REGION Network 6
   RUNG wire#powerrail
      Contact( #calcula )
      wire#w1
      { S7_Templates := "SrcType := Real"; S7_GenerateENO := "TRUE" } Sub(in1 := #FATOR, in2 := #SETPOINT, out => #FATOR)
   END_RUNG
   RUNG wire#w1
      { S7_Templates := "SrcType := Real"; S7_GenerateENO := "TRUE" } Div(in1 := #FATOR, in2 := #SETPOINT, out => #FATOR)
   END_RUNG
   RUNG wire#w1
      { S7_Templates := "SrcType := Real"; S7_GenerateENO := "TRUE" } Mul(in1 := #FATOR, in2 := #COR_MAX, out => #FATOR)
      { S7_Templates := "SrcType := Real"; S7_GenerateENO := "TRUE" } Mul(in1 := #FATOR, in2 := 0.01, out => #FATOR)
      { S7_Templates := "SrcType := Real"; S7_GenerateENO := "TRUE" } Mul(in1 := #FATOR, in2 := #VELOCIDADE_BASE, out => #CORRECAO)
   END_RUNG
   // the same network as SCL:
   // ENO of a box is taken as its EN; it also drops when the box reports an error
   IF #calcula THEN
       #FATOR := #FATOR - #SETPOINT;
       #FATOR := #FATOR / #SETPOINT;
       #FATOR := #FATOR * #COR_MAX;
       #FATOR := #FATOR * 0.01;
       #CORRECAO := #FATOR * #VELOCIDADE_BASE;
   END_IF;
END_REGION
END_FUNCTION_BLOCK

FUNCTION "GRUPO1" : Void   // FC2, LAD
{ S7_Optimized_Access := 'FALSE' }
VERSION : 0.1
   VAR_TEMP
      RASQ_R : Real;
      RASQ_DI : DInt;
      RASQ_R2 : Real;
   END_VAR
   VAR_TEMP   // added for the SCL form of the ladder/FBD networks
      _w1 : Bool;
      _w2 : Bool;
      _w3 : Bool;
      _w4 : Bool;
      _w5 : Bool;
      _w6 : Bool;
      _w7 : Bool;
      _w8 : Bool;
   END_VAR
BEGIN

REGION Network 1: RESET ALARMES
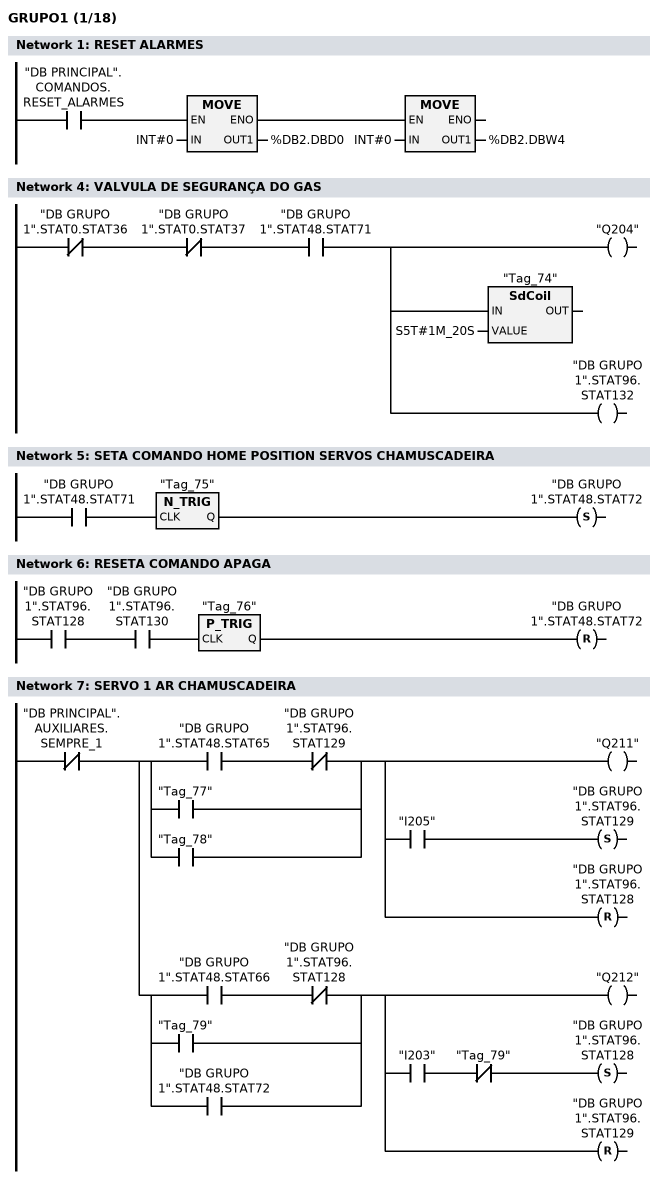
   RUNG wire#powerrail
      Contact( "DB PRINCIPAL".COMANDOS.RESET_ALARMES )
      { S7_GenerateENO := "TRUE" } Move(in := INT#0, out1 => %DB2.DBD0)
      { S7_GenerateENO := "TRUE" } Move(in := INT#0, out1 => %DB2.DBW4)
   END_RUNG
   // the same network as SCL:
   // ENO of a box is taken as its EN; it also drops when the box reports an error
   IF "DB PRINCIPAL".COMANDOS.RESET_ALARMES THEN
       %DB2.DBD0 := INT#0;
       %DB2.DBW4 := INT#0;
   END_IF;
END_REGION

REGION Network 2 (STL): TERMICOS
         A     "DB PRINCIPAL".AUXILIARES.SEMPRE_1;
         S     <??.?>;
         A     <??.?>;
         A     "I102";
         S     "DB GRUPO 1".STAT0.STAT5;
         A     <??.?>;
         A     "I103";
         S     "DB GRUPO 1".STAT0.STAT6;
         A     <??.?>;
         A     "I104";
         S     "DB GRUPO 1".STAT0.STAT7;
         A     <??.?>;
         A     "I105";
         S     "DB GRUPO 1".STAT0.STAT8;
         A     <??.?>;
         A     "I107";
         S     "DB GRUPO 1".STAT0.STAT17;
         A     <??.?>;
         A     "I110";
         S     "DB GRUPO 1".STAT0.STAT18;
         A     <??.?>;
         A     "I122";
         S     "DB GRUPO 1".STAT0.STAT19;
         A     <??.?>;
         A     "I123";
         S     "DB GRUPO 1".STAT0.STAT20;
         A     <??.?>;
         AN    "I124";
         A     "DB GRUPO 1".STAT48.STAT71;
         S     "DB GRUPO 1".STAT0.STAT3;
         A     <??.?>;
         AN    "I125";
         A     "DB GRUPO 1".STAT48.STAT71;
         S     "DB GRUPO 1".STAT0.STAT4;
         A     <??.?>;
         A     "I126";
         S     "DB GRUPO 1".STAT0.STAT10;
         A     <??.?>;
         A     "I127";
         S     "DB GRUPO 1".STAT0.STAT11;
         A     <??.?>;
         A     "I131";
         S     "DB GRUPO 1".STAT0.STAT21;
         A     <??.?>;
         A     "I133";
         S     "DB GRUPO 1".STAT0.STAT22;
         A     <??.?>;
         A     "I135";
         S     "DB GRUPO 1".STAT0.STAT23;
         A     <??.?>;
         A     "I137";
         S     "DB GRUPO 1".STAT0.STAT24;
         A     <??.?>;
         A     "I106";
         A     "DB GRUPO 1".STAT48.STAT71;
         S     "DB GRUPO 1".STAT0.STAT9;
         A     <??.?>;
         AN    "I322";
         S     "DB GRUPO 1".STAT0.STAT25;
END_REGION

REGION Network 3 (STL): ALARMES CHAMUSCADEIRA
         A     "DB GRUPO 1".STAT48.STAT71;
         =     <??.?>;
         A     <??.?>;
         AN    "I200";
         A     "Tag_72";
         S     "DB GRUPO 1".STAT0.STAT33;
         A     <??.?>;
         AN    "I207";
         A     "Tag_73";
         S     "DB GRUPO 1".STAT0.STAT38;
         A     <??.?>;
         AN    "I201";
         S     "DB GRUPO 1".STAT0.STAT34;
         A     <??.?>;
         A     "I202";
         A     "Tag_74";
         S     "DB GRUPO 1".STAT0.STAT35;
         A     <??.?>;
         AN    "I204";
         S     "DB GRUPO 1".STAT0.STAT36;
         A     <??.?>;
         A     "DB PRINCIPAL".AUXILIARES.SEMPRE_0;
         AN    "I206";
         S     "DB GRUPO 1".STAT0.STAT37;
         A     <??.?>;
         A(;
         L     "DB GRUPO 1".STAT154.STAT162;
         L     "DB GRUPO 1".STAT138.STAT146;
         >R;
         );
         S     "DB GRUPO 1".STAT0.STAT39;
         A     <??.?>;
         A(;
         L     "DB GRUPO 1".STAT154.STAT163;
         L     "DB GRUPO 1".STAT138.STAT147;
         >R;
         );
         S     "DB GRUPO 1".STAT0.STAT40;
         A     <??.?>;
         A(;
         L     "DB GRUPO 1".STAT154.STAT164;
         L     "DB GRUPO 1".STAT138.STAT148;
         >R;
         );
         S     "DB GRUPO 1".STAT0.STAT41;
         A     <??.?>;
         A(;
         L     "DB GRUPO 1".STAT154.STAT165;
         L     "DB GRUPO 1".STAT138.STAT149;
         >R;
         );
         S     "DB GRUPO 1".STAT0.STAT42;
         A     <??.?>;
         A     "I214";
         S     "DB GRUPO 1".STAT0.STAT43;
         A     <??.?>;
         A     "I215";
         S     "DB GRUPO 1".STAT0.STAT44;
         A     <??.?>;
         A     "I216";
         S     "DB GRUPO 1".STAT0.STAT45;
         A     <??.?>;
         A     "I217";
         S     "DB GRUPO 1".STAT0.STAT46;
         NOP   0;
END_REGION

REGION Network 4: VALVULA DE SEGURANÇA DO GAS
   // no SCL statement known for SdCoil: written as a call
   "Q204" := NOT "DB GRUPO 1".STAT0.STAT36 AND NOT "DB GRUPO 1".STAT0.STAT37 AND "DB GRUPO 1".STAT48.STAT71;
   #_w1 := "Q204";
   SdCoil(value := S5T#1M_20S, operand := "Tag_74", in := "Q204");
   "DB GRUPO 1".STAT96.STAT132 := #_w1;
END_REGION

REGION Network 5: SETA COMANDO HOME POSITION SERVOS CHAMUSCADEIRA
   RUNG wire#powerrail
      Contact( "DB GRUPO 1".STAT48.STAT71 )
      N_Trig( "Tag_75" )
      S_Coil( "DB GRUPO 1".STAT48.STAT72 )
   END_RUNG
   // the same network as SCL:
   #_w1 := NOT "DB GRUPO 1".STAT48.STAT71 AND "Tag_75";   // falling edge
   "Tag_75" := "DB GRUPO 1".STAT48.STAT71;
   IF #_w1 THEN "DB GRUPO 1".STAT48.STAT72 := TRUE; END_IF;
END_REGION

REGION Network 6: RESETA COMANDO APAGA
   RUNG wire#powerrail
      Contact( "DB GRUPO 1".STAT96.STAT128 )
      Contact( "DB GRUPO 1".STAT96.STAT130 )
      P_Trig( "Tag_76" )
      R_Coil( "DB GRUPO 1".STAT48.STAT72 )
   END_RUNG
   // the same network as SCL:
   #_w1 := "DB GRUPO 1".STAT96.STAT128 AND "DB GRUPO 1".STAT96.STAT130;
   #_w2 := #_w1 AND NOT "Tag_76";   // rising edge
   "Tag_76" := #_w1;
   IF #_w2 THEN "DB GRUPO 1".STAT48.STAT72 := FALSE; END_IF;
END_REGION

REGION Network 7: SERVO 1 AR CHAMUSCADEIRA
   RUNG wire#powerrail
      I_Contact( "DB PRINCIPAL".AUXILIARES.SEMPRE_1 )
      wire#w1
      Contact( "DB GRUPO 1".STAT48.STAT65 )
      I_Contact( "DB GRUPO 1".STAT96.STAT129 )
      wire#w2
      Coil( "Q211" )
   END_RUNG
   RUNG wire#w1
      Contact( "Tag_77" )
   END_RUNG wire#w2
   RUNG wire#w1
      Contact( "Tag_78" )
   END_RUNG wire#w2
   RUNG wire#w2
      Contact( "I205" )
      S_Coil( "DB GRUPO 1".STAT96.STAT129 )
   END_RUNG
   RUNG wire#w2
      R_Coil( "DB GRUPO 1".STAT96.STAT128 )
   END_RUNG
   RUNG wire#w1
      Contact( "DB GRUPO 1".STAT48.STAT66 )
      I_Contact( "DB GRUPO 1".STAT96.STAT128 )
      wire#w3
      Coil( "Q212" )
   END_RUNG
   RUNG wire#w1
      Contact( "Tag_79" )
   END_RUNG wire#w3
   RUNG wire#w1
      Contact( "DB GRUPO 1".STAT48.STAT72 )
   END_RUNG wire#w3
   RUNG wire#w3
      Contact( "I203" )
      I_Contact( "Tag_79" )
      S_Coil( "DB GRUPO 1".STAT96.STAT128 )
   END_RUNG
   RUNG wire#w3
      R_Coil( "DB GRUPO 1".STAT96.STAT129 )
   END_RUNG
   // the same network as SCL:
   #_w1 := NOT "DB PRINCIPAL".AUXILIARES.SEMPRE_1;
   "Q211" := #_w1 AND (("DB GRUPO 1".STAT48.STAT65 AND NOT "DB GRUPO 1".STAT96.STAT129) OR "Tag_77" OR "Tag_78");
   IF "Q211" AND "I205" THEN "DB GRUPO 1".STAT96.STAT129 := TRUE; END_IF;
   IF "Q211" THEN "DB GRUPO 1".STAT96.STAT128 := FALSE; END_IF;
   "Q212" := #_w1 AND (("DB GRUPO 1".STAT48.STAT66 AND NOT "DB GRUPO 1".STAT96.STAT128) OR "Tag_79" OR "DB GRUPO 1".STAT48.STAT72);
   IF "Q212" AND "I203" AND NOT "Tag_79" THEN "DB GRUPO 1".STAT96.STAT128 := TRUE; END_IF;
   IF "Q212" THEN "DB GRUPO 1".STAT96.STAT129 := FALSE; END_IF;
END_REGION

REGION Network 8: SERVO 2 AR CHAMUSCADEIRA
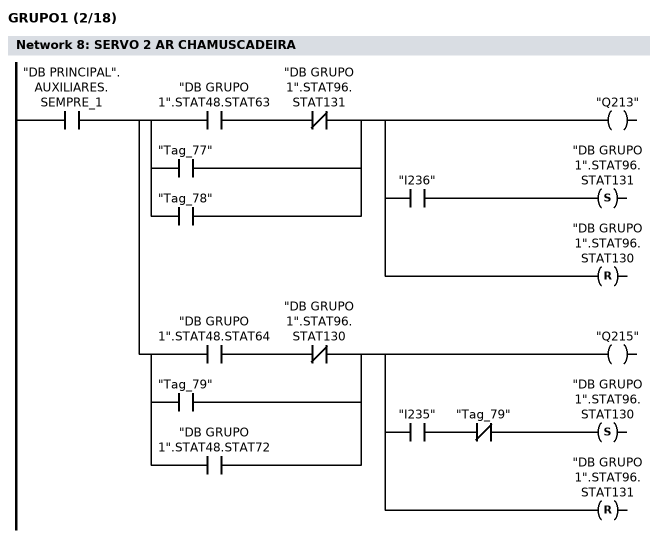
   RUNG wire#powerrail
      Contact( "DB PRINCIPAL".AUXILIARES.SEMPRE_1 )
      wire#w1
      Contact( "DB GRUPO 1".STAT48.STAT63 )
      I_Contact( "DB GRUPO 1".STAT96.STAT131 )
      wire#w2
      Coil( "Q213" )
   END_RUNG
   RUNG wire#w1
      Contact( "Tag_77" )
   END_RUNG wire#w2
   RUNG wire#w1
      Contact( "Tag_78" )
   END_RUNG wire#w2
   RUNG wire#w2
      Contact( "I236" )
      S_Coil( "DB GRUPO 1".STAT96.STAT131 )
   END_RUNG
   RUNG wire#w2
      R_Coil( "DB GRUPO 1".STAT96.STAT130 )
   END_RUNG
   RUNG wire#w1
      Contact( "DB GRUPO 1".STAT48.STAT64 )
      I_Contact( "DB GRUPO 1".STAT96.STAT130 )
      wire#w3
      Coil( "Q215" )
   END_RUNG
   RUNG wire#w1
      Contact( "Tag_79" )
   END_RUNG wire#w3
   RUNG wire#w1
      Contact( "DB GRUPO 1".STAT48.STAT72 )
   END_RUNG wire#w3
   RUNG wire#w3
      Contact( "I235" )
      I_Contact( "Tag_79" )
      S_Coil( "DB GRUPO 1".STAT96.STAT130 )
   END_RUNG
   RUNG wire#w3
      R_Coil( "DB GRUPO 1".STAT96.STAT131 )
   END_RUNG
   // the same network as SCL:
   "Q213" := "DB PRINCIPAL".AUXILIARES.SEMPRE_1 AND (("DB GRUPO 1".STAT48.STAT63 AND NOT "DB GRUPO 1".STAT96.STAT131) OR "Tag_77" OR "Tag_78");
   IF "Q213" AND "I236" THEN "DB GRUPO 1".STAT96.STAT131 := TRUE; END_IF;
   IF "Q213" THEN "DB GRUPO 1".STAT96.STAT130 := FALSE; END_IF;
   "Q215" := "DB PRINCIPAL".AUXILIARES.SEMPRE_1 AND (("DB GRUPO 1".STAT48.STAT64 AND NOT "DB GRUPO 1".STAT96.STAT130) OR "Tag_79" OR "DB GRUPO 1".STAT48.STAT72);
   IF "Q215" AND "I235" AND NOT "Tag_79" THEN "DB GRUPO 1".STAT96.STAT130 := TRUE; END_IF;
   IF "Q215" THEN "DB GRUPO 1".STAT96.STAT131 := FALSE; END_IF;
END_REGION

REGION Network 9: COMANDA POSIÇÃO DA CHAMA
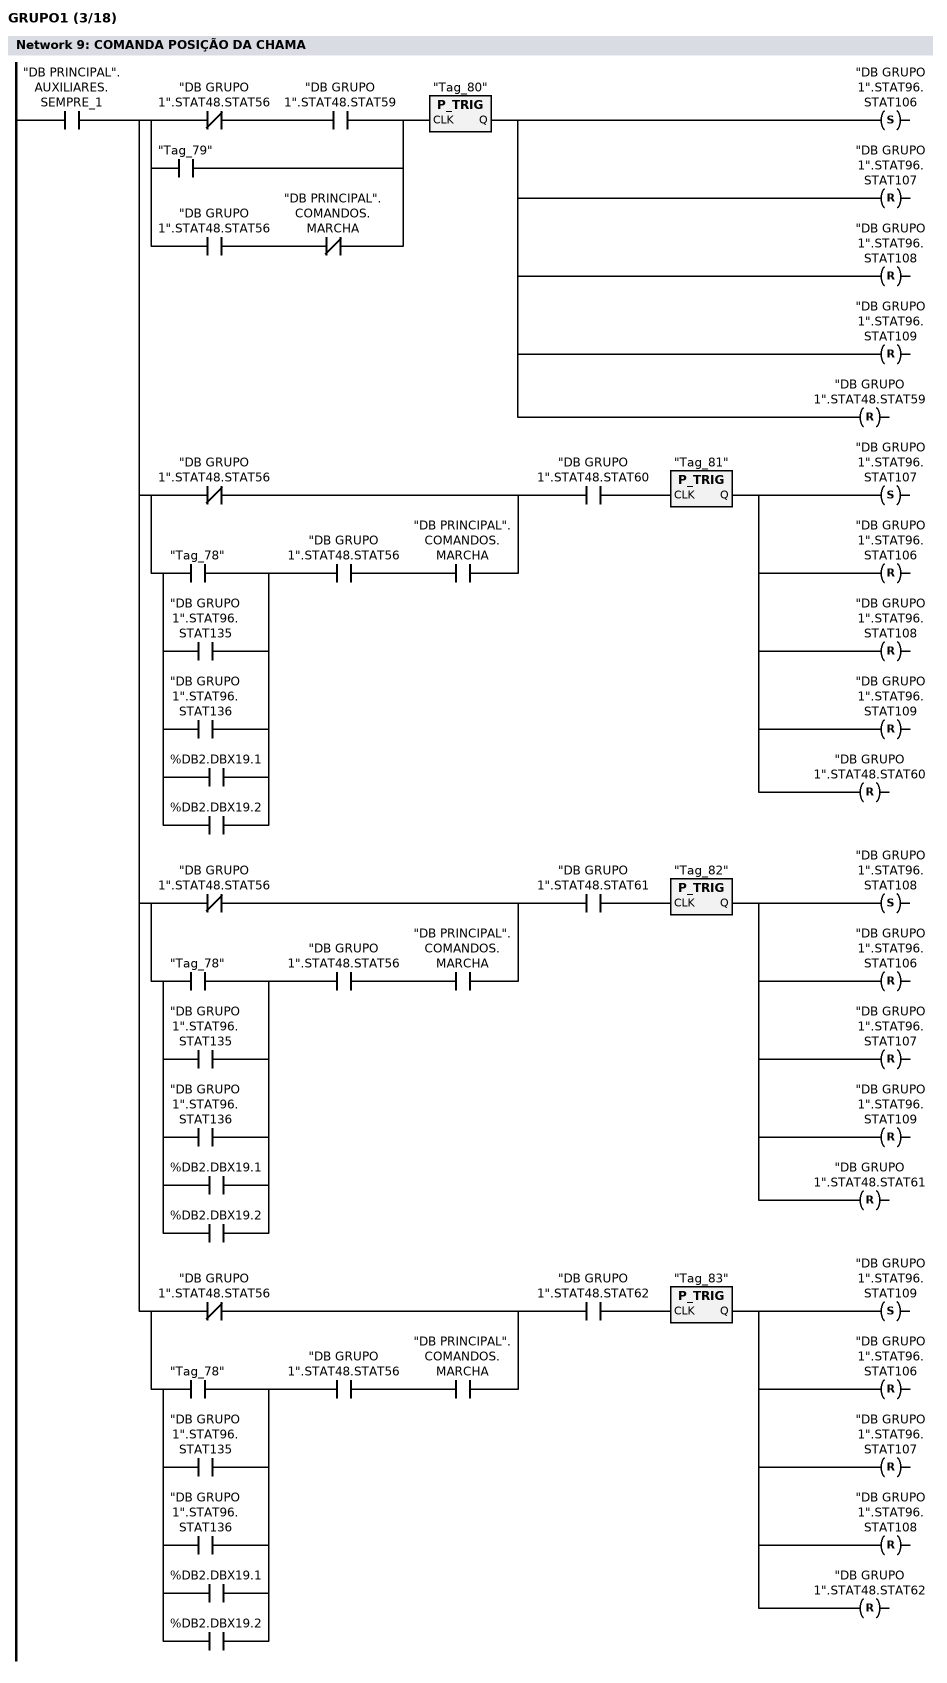
   RUNG wire#powerrail
      Contact( "DB PRINCIPAL".AUXILIARES.SEMPRE_1 )
      wire#w1
      I_Contact( "DB GRUPO 1".STAT48.STAT56 )
      Contact( "DB GRUPO 1".STAT48.STAT59 )
      wire#w2
      P_Trig( "Tag_80" )
      wire#w3
      S_Coil( "DB GRUPO 1".STAT96.STAT106 )
   END_RUNG
   RUNG wire#w1
      Contact( "Tag_79" )
   END_RUNG wire#w2
   RUNG wire#w1
      Contact( "DB GRUPO 1".STAT48.STAT56 )
      I_Contact( "DB PRINCIPAL".COMANDOS.MARCHA )
   END_RUNG wire#w2
   RUNG wire#w3
      R_Coil( "DB GRUPO 1".STAT96.STAT107 )
   END_RUNG
   RUNG wire#w3
      R_Coil( "DB GRUPO 1".STAT96.STAT108 )
   END_RUNG
   RUNG wire#w3
      R_Coil( "DB GRUPO 1".STAT96.STAT109 )
   END_RUNG
   RUNG wire#w3
      R_Coil( "DB GRUPO 1".STAT48.STAT59 )
   END_RUNG
   RUNG wire#w1
      I_Contact( "DB GRUPO 1".STAT48.STAT56 )
      wire#w4
      Contact( "DB GRUPO 1".STAT48.STAT60 )
      P_Trig( "Tag_81" )
      wire#w6
      S_Coil( "DB GRUPO 1".STAT96.STAT107 )
   END_RUNG
   RUNG wire#w1
      Contact( "Tag_78" )
      wire#w5
      Contact( "DB GRUPO 1".STAT48.STAT56 )
      Contact( "DB PRINCIPAL".COMANDOS.MARCHA )
   END_RUNG wire#w4
   RUNG wire#w1
      Contact( "DB GRUPO 1".STAT96.STAT135 )
   END_RUNG wire#w5
   RUNG wire#w1
      Contact( "DB GRUPO 1".STAT96.STAT136 )
   END_RUNG wire#w5
   RUNG wire#w1
      Contact( %DB2.DBX19.1 )
   END_RUNG wire#w5
   RUNG wire#w1
      Contact( %DB2.DBX19.2 )
   END_RUNG wire#w5
   RUNG wire#w6
      R_Coil( "DB GRUPO 1".STAT96.STAT106 )
   END_RUNG
   RUNG wire#w6
      R_Coil( "DB GRUPO 1".STAT96.STAT108 )
   END_RUNG
   RUNG wire#w6
      R_Coil( "DB GRUPO 1".STAT96.STAT109 )
   END_RUNG
   RUNG wire#w6
      R_Coil( "DB GRUPO 1".STAT48.STAT60 )
   END_RUNG
   RUNG wire#w1
      I_Contact( "DB GRUPO 1".STAT48.STAT56 )
      wire#w7
      Contact( "DB GRUPO 1".STAT48.STAT61 )
      P_Trig( "Tag_82" )
      wire#w9
      S_Coil( "DB GRUPO 1".STAT96.STAT108 )
   END_RUNG
   RUNG wire#w1
      Contact( "Tag_78" )
      wire#w8
      Contact( "DB GRUPO 1".STAT48.STAT56 )
      Contact( "DB PRINCIPAL".COMANDOS.MARCHA )
   END_RUNG wire#w7
   RUNG wire#w1
      Contact( "DB GRUPO 1".STAT96.STAT135 )
   END_RUNG wire#w8
   RUNG wire#w1
      Contact( "DB GRUPO 1".STAT96.STAT136 )
   END_RUNG wire#w8
   RUNG wire#w1
      Contact( %DB2.DBX19.1 )
   END_RUNG wire#w8
   RUNG wire#w1
      Contact( %DB2.DBX19.2 )
   END_RUNG wire#w8
   RUNG wire#w9
      R_Coil( "DB GRUPO 1".STAT96.STAT106 )
   END_RUNG
   RUNG wire#w9
      R_Coil( "DB GRUPO 1".STAT96.STAT107 )
   END_RUNG
   RUNG wire#w9
      R_Coil( "DB GRUPO 1".STAT96.STAT109 )
   END_RUNG
   RUNG wire#w9
      R_Coil( "DB GRUPO 1".STAT48.STAT61 )
   END_RUNG
   RUNG wire#w1
      I_Contact( "DB GRUPO 1".STAT48.STAT56 )
      wire#w10
      Contact( "DB GRUPO 1".STAT48.STAT62 )
      P_Trig( "Tag_83" )
      wire#w12
      S_Coil( "DB GRUPO 1".STAT96.STAT109 )
   END_RUNG
   RUNG wire#w1
      Contact( "Tag_78" )
      wire#w11
      Contact( "DB GRUPO 1".STAT48.STAT56 )
      Contact( "DB PRINCIPAL".COMANDOS.MARCHA )
   END_RUNG wire#w10
   RUNG wire#w1
      Contact( "DB GRUPO 1".STAT96.STAT135 )
   END_RUNG wire#w11
   RUNG wire#w1
      Contact( "DB GRUPO 1".STAT96.STAT136 )
   END_RUNG wire#w11
   RUNG wire#w1
      Contact( %DB2.DBX19.1 )
   END_RUNG wire#w11
   RUNG wire#w1
      Contact( %DB2.DBX19.2 )
   END_RUNG wire#w11
   RUNG wire#w12
      R_Coil( "DB GRUPO 1".STAT96.STAT106 )
   END_RUNG
   RUNG wire#w12
      R_Coil( "DB GRUPO 1".STAT96.STAT107 )
   END_RUNG
   RUNG wire#w12
      R_Coil( "DB GRUPO 1".STAT96.STAT108 )
   END_RUNG
   RUNG wire#w12
      R_Coil( "DB GRUPO 1".STAT48.STAT62 )
   END_RUNG
   // the same network as SCL:
   #_w1 := "DB PRINCIPAL".AUXILIARES.SEMPRE_1 AND ((NOT "DB GRUPO 1".STAT48.STAT56 AND "DB GRUPO 1".STAT48.STAT59) OR "Tag_79" OR ("DB GRUPO 1".STAT48.STAT56 AND NOT "DB PRINCIPAL".COMANDOS.MARCHA));
   #_w2 := #_w1 AND NOT "Tag_80";   // rising edge
   "Tag_80" := #_w1;
   IF #_w2 THEN
       "DB GRUPO 1".STAT96.STAT106 := TRUE;
       "DB GRUPO 1".STAT96.STAT107 := FALSE;
       "DB GRUPO 1".STAT96.STAT108 := FALSE;
       "DB GRUPO 1".STAT96.STAT109 := FALSE;
       "DB GRUPO 1".STAT48.STAT59 := FALSE;
   END_IF;
   #_w3 := "DB PRINCIPAL".AUXILIARES.SEMPRE_1 AND (NOT "DB GRUPO 1".STAT48.STAT56 OR (("Tag_78" OR "DB GRUPO 1".STAT96.STAT135 OR "DB GRUPO 1".STAT96.STAT136 OR %DB2.DBX19.1 OR %DB2.DBX19.2) AND "DB GRUPO 1".STAT48.STAT56 AND "DB PRINCIPAL".COMANDOS.MARCHA)) AND "DB GRUPO 1".STAT48.STAT60;
   #_w4 := #_w3 AND NOT "Tag_81";   // rising edge
   "Tag_81" := #_w3;
   IF #_w4 THEN
       "DB GRUPO 1".STAT96.STAT107 := TRUE;
       "DB GRUPO 1".STAT96.STAT106 := FALSE;
       "DB GRUPO 1".STAT96.STAT108 := FALSE;
       "DB GRUPO 1".STAT96.STAT109 := FALSE;
       "DB GRUPO 1".STAT48.STAT60 := FALSE;
   END_IF;
   #_w5 := "DB PRINCIPAL".AUXILIARES.SEMPRE_1 AND (NOT "DB GRUPO 1".STAT48.STAT56 OR (("Tag_78" OR "DB GRUPO 1".STAT96.STAT135 OR "DB GRUPO 1".STAT96.STAT136 OR %DB2.DBX19.1 OR %DB2.DBX19.2) AND "DB GRUPO 1".STAT48.STAT56 AND "DB PRINCIPAL".COMANDOS.MARCHA)) AND "DB GRUPO 1".STAT48.STAT61;
   #_w6 := #_w5 AND NOT "Tag_82";   // rising edge
   "Tag_82" := #_w5;
   IF #_w6 THEN
       "DB GRUPO 1".STAT96.STAT108 := TRUE;
       "DB GRUPO 1".STAT96.STAT106 := FALSE;
       "DB GRUPO 1".STAT96.STAT107 := FALSE;
       "DB GRUPO 1".STAT96.STAT109 := FALSE;
       "DB GRUPO 1".STAT48.STAT61 := FALSE;
   END_IF;
   #_w7 := "DB PRINCIPAL".AUXILIARES.SEMPRE_1 AND (NOT "DB GRUPO 1".STAT48.STAT56 OR (("Tag_78" OR "DB GRUPO 1".STAT96.STAT135 OR "DB GRUPO 1".STAT96.STAT136 OR %DB2.DBX19.1 OR %DB2.DBX19.2) AND "DB GRUPO 1".STAT48.STAT56 AND "DB PRINCIPAL".COMANDOS.MARCHA)) AND "DB GRUPO 1".STAT48.STAT62;
   #_w8 := #_w7 AND NOT "Tag_83";   // rising edge
   "Tag_83" := #_w7;
   IF #_w8 THEN
       "DB GRUPO 1".STAT96.STAT109 := TRUE;
       "DB GRUPO 1".STAT96.STAT106 := FALSE;
       "DB GRUPO 1".STAT96.STAT107 := FALSE;
       "DB GRUPO 1".STAT96.STAT108 := FALSE;
       "DB GRUPO 1".STAT48.STAT62 := FALSE;
   END_IF;
END_REGION

REGION Network 10: POSICIONA A CHAMA
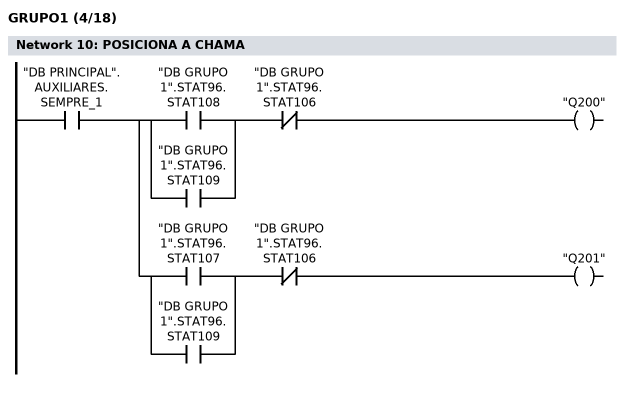
   RUNG wire#powerrail
      Contact( "DB PRINCIPAL".AUXILIARES.SEMPRE_1 )
      wire#w1
      Contact( "DB GRUPO 1".STAT96.STAT108 )
      wire#w2
      I_Contact( "DB GRUPO 1".STAT96.STAT106 )
      Coil( "Q200" )
   END_RUNG
   RUNG wire#w1
      Contact( "DB GRUPO 1".STAT96.STAT109 )
   END_RUNG wire#w2
   RUNG wire#w1
      Contact( "DB GRUPO 1".STAT96.STAT107 )
      wire#w3
      I_Contact( "DB GRUPO 1".STAT96.STAT106 )
      Coil( "Q201" )
   END_RUNG
   RUNG wire#w1
      Contact( "DB GRUPO 1".STAT96.STAT109 )
   END_RUNG wire#w3
   // the same network as SCL:
   "Q200" := "DB PRINCIPAL".AUXILIARES.SEMPRE_1 AND ("DB GRUPO 1".STAT96.STAT108 OR "DB GRUPO 1".STAT96.STAT109) AND NOT "DB GRUPO 1".STAT96.STAT106;
   "Q201" := "DB PRINCIPAL".AUXILIARES.SEMPRE_1 AND ("DB GRUPO 1".STAT96.STAT107 OR "DB GRUPO 1".STAT96.STAT109) AND NOT "DB GRUPO 1".STAT96.STAT106;
END_REGION

REGION Network 11: ACENDIMENTO MANUAL OU AUTOMATICO
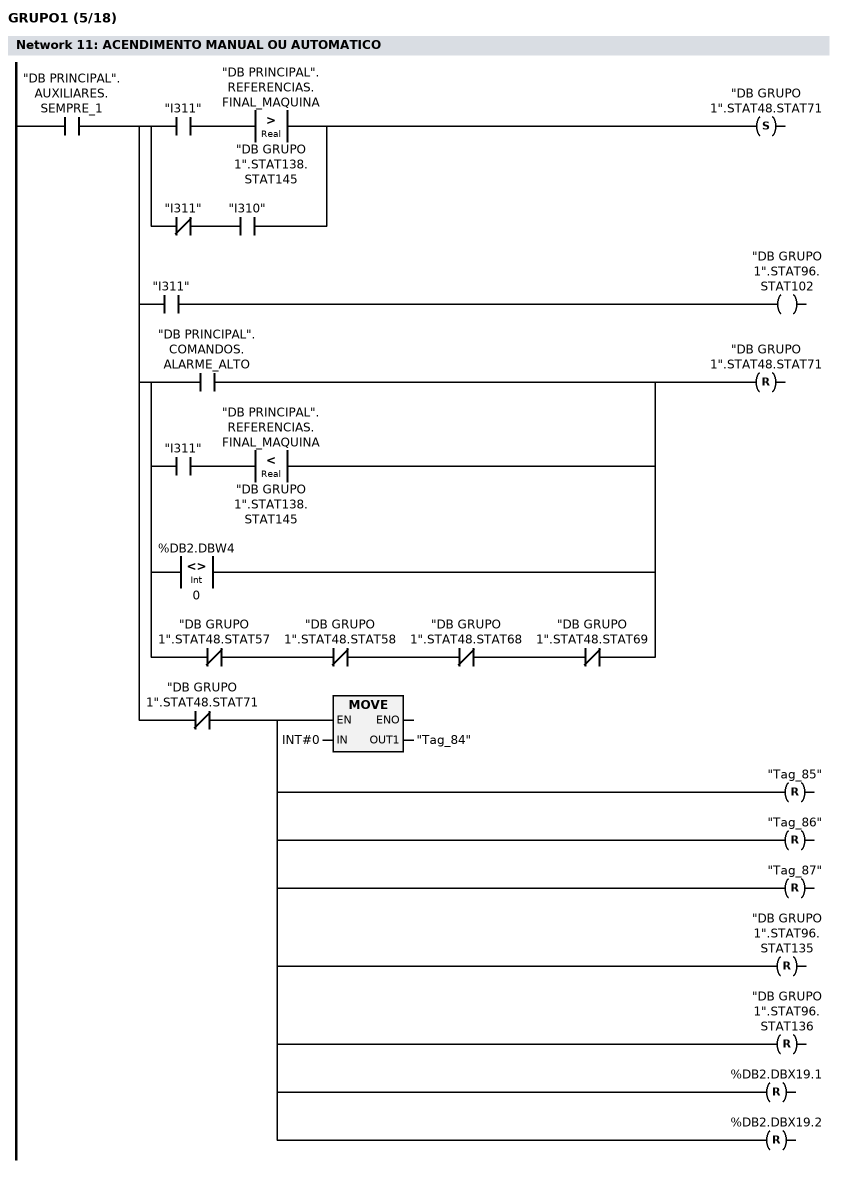
   IF "DB PRINCIPAL".AUXILIARES.SEMPRE_1 AND (("I311" AND ("DB PRINCIPAL".REFERENCIAS.FINAL_MAQUINA > "DB GRUPO 1".STAT138.STAT145)) OR (NOT "I311" AND "I310")) THEN
       "DB GRUPO 1".STAT48.STAT71 := TRUE;
   END_IF;
   "DB GRUPO 1".STAT96.STAT102 := "DB PRINCIPAL".AUXILIARES.SEMPRE_1 AND "I311";
   IF "DB PRINCIPAL".AUXILIARES.SEMPRE_1 AND (("I311" AND ("DB PRINCIPAL".REFERENCIAS.FINAL_MAQUINA < "DB GRUPO 1".STAT138.STAT145)) OR (%DB2.DBW4 <> 0) OR "DB PRINCIPAL".COMANDOS.ALARME_ALTO OR (NOT "DB GRUPO 1".STAT48.STAT57 AND NOT "DB GRUPO 1".STAT48.STAT58 AND NOT "DB GRUPO 1".STAT48.STAT68 AND NOT "DB GRUPO 1".STAT48.STAT69)) THEN
       "DB GRUPO 1".STAT48.STAT71 := FALSE;
   END_IF;
   IF "DB PRINCIPAL".AUXILIARES.SEMPRE_1 AND NOT "DB GRUPO 1".STAT48.STAT71 THEN
       "Tag_84" := INT#0;
       "Tag_85" := FALSE;
       "Tag_86" := FALSE;
       "Tag_87" := FALSE;
       "DB GRUPO 1".STAT96.STAT135 := FALSE;
       "DB GRUPO 1".STAT96.STAT136 := FALSE;
       %DB2.DBX19.1 := FALSE;
       %DB2.DBX19.2 := FALSE;
   END_IF;
END_REGION

REGION Network 12: STATUS DAS CHAMAS DOS QUEIMADORES
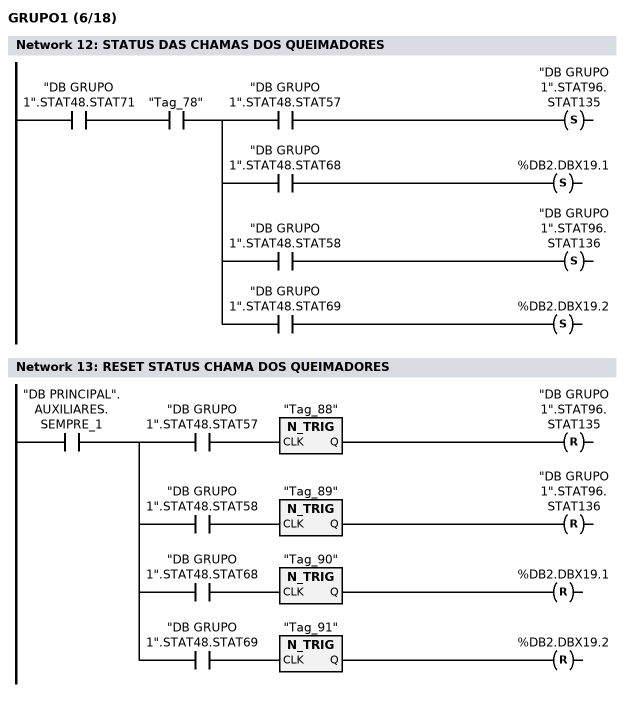
   RUNG wire#powerrail
      Contact( "DB GRUPO 1".STAT48.STAT71 )
      Contact( "Tag_78" )
      wire#w1
      Contact( "DB GRUPO 1".STAT48.STAT57 )
      S_Coil( "DB GRUPO 1".STAT96.STAT135 )
   END_RUNG
   RUNG wire#w1
      Contact( "DB GRUPO 1".STAT48.STAT68 )
      S_Coil( %DB2.DBX19.1 )
   END_RUNG
   RUNG wire#w1
      Contact( "DB GRUPO 1".STAT48.STAT58 )
      S_Coil( "DB GRUPO 1".STAT96.STAT136 )
   END_RUNG
   RUNG wire#w1
      Contact( "DB GRUPO 1".STAT48.STAT69 )
      S_Coil( %DB2.DBX19.2 )
   END_RUNG
   // the same network as SCL:
   #_w1 := "DB GRUPO 1".STAT48.STAT71 AND "Tag_78";
   IF #_w1 AND "DB GRUPO 1".STAT48.STAT57 THEN "DB GRUPO 1".STAT96.STAT135 := TRUE; END_IF;
   IF #_w1 AND "DB GRUPO 1".STAT48.STAT68 THEN %DB2.DBX19.1 := TRUE; END_IF;
   IF #_w1 AND "DB GRUPO 1".STAT48.STAT58 THEN "DB GRUPO 1".STAT96.STAT136 := TRUE; END_IF;
   IF #_w1 AND "DB GRUPO 1".STAT48.STAT69 THEN %DB2.DBX19.2 := TRUE; END_IF;
END_REGION

REGION Network 13: RESET STATUS CHAMA DOS QUEIMADORES
   RUNG wire#powerrail
      Contact( "DB PRINCIPAL".AUXILIARES.SEMPRE_1 )
      wire#w1
      Contact( "DB GRUPO 1".STAT48.STAT57 )
      N_Trig( "Tag_88" )
      R_Coil( "DB GRUPO 1".STAT96.STAT135 )
   END_RUNG
   RUNG wire#w1
      Contact( "DB GRUPO 1".STAT48.STAT58 )
      N_Trig( "Tag_89" )
      R_Coil( "DB GRUPO 1".STAT96.STAT136 )
   END_RUNG
   RUNG wire#w1
      Contact( "DB GRUPO 1".STAT48.STAT68 )
      N_Trig( "Tag_90" )
      R_Coil( %DB2.DBX19.1 )
   END_RUNG
   RUNG wire#w1
      Contact( "DB GRUPO 1".STAT48.STAT69 )
      N_Trig( "Tag_91" )
      R_Coil( %DB2.DBX19.2 )
   END_RUNG
   // the same network as SCL:
   #_w1 := "DB PRINCIPAL".AUXILIARES.SEMPRE_1 AND "DB GRUPO 1".STAT48.STAT57;
   #_w2 := NOT #_w1 AND "Tag_88";   // falling edge
   "Tag_88" := #_w1;
   IF #_w2 THEN "DB GRUPO 1".STAT96.STAT135 := FALSE; END_IF;
   #_w3 := "DB PRINCIPAL".AUXILIARES.SEMPRE_1 AND "DB GRUPO 1".STAT48.STAT58;
   #_w4 := NOT #_w3 AND "Tag_89";   // falling edge
   "Tag_89" := #_w3;
   IF #_w4 THEN "DB GRUPO 1".STAT96.STAT136 := FALSE; END_IF;
   #_w5 := "DB PRINCIPAL".AUXILIARES.SEMPRE_1 AND "DB GRUPO 1".STAT48.STAT68;
   #_w6 := NOT #_w5 AND "Tag_90";   // falling edge
   "Tag_90" := #_w5;
   IF #_w6 THEN %DB2.DBX19.1 := FALSE; END_IF;
   #_w7 := "DB PRINCIPAL".AUXILIARES.SEMPRE_1 AND "DB GRUPO 1".STAT48.STAT69;
   #_w8 := NOT #_w7 AND "Tag_91";   // falling edge
   "Tag_91" := #_w7;
   IF #_w8 THEN %DB2.DBX19.2 := FALSE; END_IF;
END_REGION

REGION Network 14: SEQUENCIA DE ACENDIMENTO DA CHAMUSCADEIRA
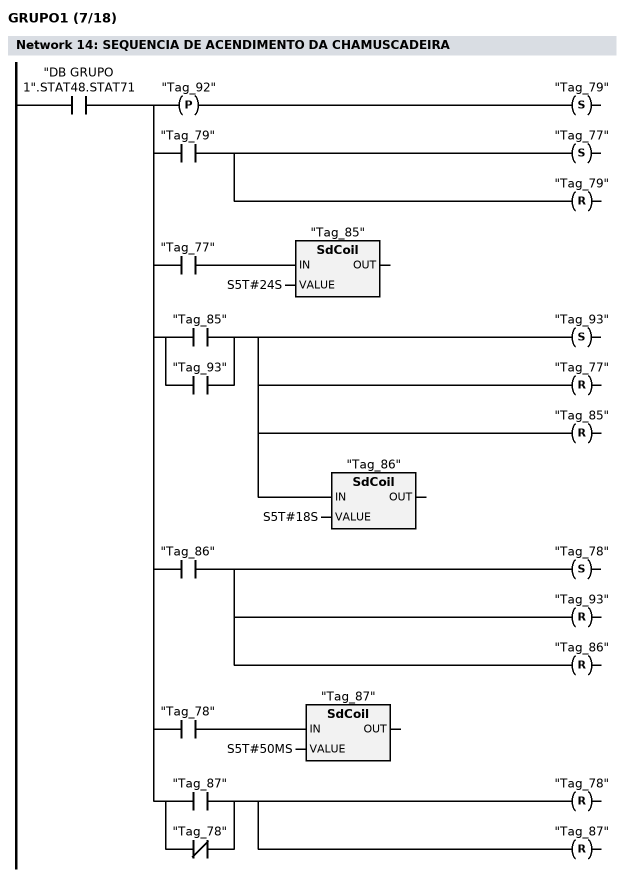
   // no SCL statement known for SdCoil: written as a call
   #_w1 := "DB GRUPO 1".STAT48.STAT71 AND NOT "Tag_92";   // rising edge
   "Tag_92" := "DB GRUPO 1".STAT48.STAT71;
   IF #_w1 THEN "Tag_79" := TRUE; END_IF;
   IF "DB GRUPO 1".STAT48.STAT71 AND "Tag_79" THEN
       "Tag_77" := TRUE;
       "Tag_79" := FALSE;
   END_IF;
   #_w2 := "DB GRUPO 1".STAT48.STAT71;
   SdCoil(value := S5T#24S, operand := "Tag_85", in := "DB GRUPO 1".STAT48.STAT71 AND "Tag_77");
   #_w3 := #_w2 AND ("Tag_85" OR "Tag_93");
   IF #_w3 THEN
       "Tag_93" := TRUE;
       "Tag_77" := FALSE;
       "Tag_85" := FALSE;
   END_IF;
   SdCoil(in := #_w3, value := S5T#18S, operand := "Tag_86");
   IF #_w2 AND "Tag_86" THEN
       "Tag_78" := TRUE;
       "Tag_93" := FALSE;
       "Tag_86" := FALSE;
   END_IF;
   SdCoil(value := S5T#50MS, operand := "Tag_87", in := #_w2 AND "Tag_78");
   #_w4 := #_w2 AND ("Tag_87" OR NOT "Tag_78");
   IF #_w4 THEN
       "Tag_78" := FALSE;
       "Tag_87" := FALSE;
   END_IF;
END_REGION

REGION Network 15: CONTROLE DOS PROGRAMADORES SELCON
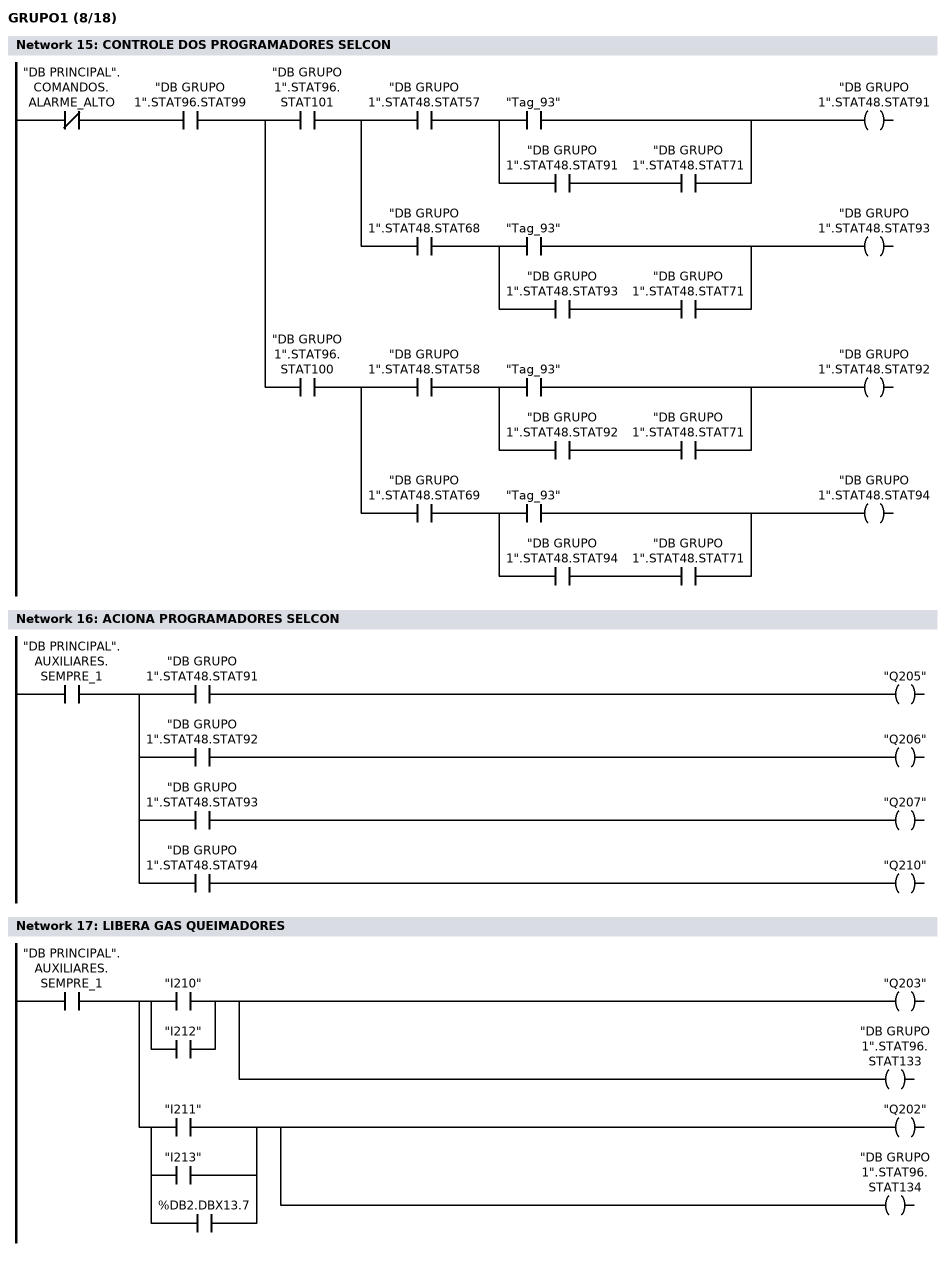
   RUNG wire#powerrail
      I_Contact( "DB PRINCIPAL".COMANDOS.ALARME_ALTO )
      Contact( "DB GRUPO 1".STAT96.STAT99 )
      wire#w1
      Contact( "DB GRUPO 1".STAT96.STAT101 )
      wire#w2
      Contact( "DB GRUPO 1".STAT48.STAT57 )
      wire#w3
      Contact( "Tag_93" )
      wire#w4
      Coil( "DB GRUPO 1".STAT48.STAT91 )
   END_RUNG
   RUNG wire#w3
      Contact( "DB GRUPO 1".STAT48.STAT91 )
      Contact( "DB GRUPO 1".STAT48.STAT71 )
   END_RUNG wire#w4
   RUNG wire#w2
      Contact( "DB GRUPO 1".STAT48.STAT68 )
      wire#w5
      Contact( "Tag_93" )
      wire#w6
      Coil( "DB GRUPO 1".STAT48.STAT93 )
   END_RUNG
   RUNG wire#w5
      Contact( "DB GRUPO 1".STAT48.STAT93 )
      Contact( "DB GRUPO 1".STAT48.STAT71 )
   END_RUNG wire#w6
   RUNG wire#w1
      Contact( "DB GRUPO 1".STAT96.STAT100 )
      wire#w7
      Contact( "DB GRUPO 1".STAT48.STAT58 )
      wire#w8
      Contact( "Tag_93" )
      wire#w9
      Coil( "DB GRUPO 1".STAT48.STAT92 )
   END_RUNG
   RUNG wire#w8
      Contact( "DB GRUPO 1".STAT48.STAT92 )
      Contact( "DB GRUPO 1".STAT48.STAT71 )
   END_RUNG wire#w9
   RUNG wire#w7
      Contact( "DB GRUPO 1".STAT48.STAT69 )
      wire#w10
      Contact( "Tag_93" )
      wire#w11
      Coil( "DB GRUPO 1".STAT48.STAT94 )
   END_RUNG
   RUNG wire#w10
      Contact( "DB GRUPO 1".STAT48.STAT94 )
      Contact( "DB GRUPO 1".STAT48.STAT71 )
   END_RUNG wire#w11
   // the same network as SCL:
   #_w1 := NOT "DB PRINCIPAL".COMANDOS.ALARME_ALTO AND "DB GRUPO 1".STAT96.STAT99;
   #_w2 := #_w1 AND "DB GRUPO 1".STAT96.STAT101;
   "DB GRUPO 1".STAT48.STAT91 := #_w2 AND "DB GRUPO 1".STAT48.STAT57 AND ("Tag_93" OR ("DB GRUPO 1".STAT48.STAT91 AND "DB GRUPO 1".STAT48.STAT71));
   "DB GRUPO 1".STAT48.STAT93 := #_w2 AND "DB GRUPO 1".STAT48.STAT68 AND ("Tag_93" OR ("DB GRUPO 1".STAT48.STAT93 AND "DB GRUPO 1".STAT48.STAT71));
   #_w3 := #_w1 AND "DB GRUPO 1".STAT96.STAT100;
   "DB GRUPO 1".STAT48.STAT92 := #_w3 AND "DB GRUPO 1".STAT48.STAT58 AND ("Tag_93" OR ("DB GRUPO 1".STAT48.STAT92 AND "DB GRUPO 1".STAT48.STAT71));
   "DB GRUPO 1".STAT48.STAT94 := #_w3 AND "DB GRUPO 1".STAT48.STAT69 AND ("Tag_93" OR ("DB GRUPO 1".STAT48.STAT94 AND "DB GRUPO 1".STAT48.STAT71));
END_REGION

REGION Network 16: ACIONA PROGRAMADORES SELCON
   RUNG wire#powerrail
      Contact( "DB PRINCIPAL".AUXILIARES.SEMPRE_1 )
      wire#w1
      Contact( "DB GRUPO 1".STAT48.STAT91 )
      Coil( "Q205" )
   END_RUNG
   RUNG wire#w1
      Contact( "DB GRUPO 1".STAT48.STAT92 )
      Coil( "Q206" )
   END_RUNG
   RUNG wire#w1
      Contact( "DB GRUPO 1".STAT48.STAT93 )
      Coil( "Q207" )
   END_RUNG
   RUNG wire#w1
      Contact( "DB GRUPO 1".STAT48.STAT94 )
      Coil( "Q210" )
   END_RUNG
   // the same network as SCL:
   "Q205" := "DB PRINCIPAL".AUXILIARES.SEMPRE_1 AND "DB GRUPO 1".STAT48.STAT91;
   "Q206" := "DB PRINCIPAL".AUXILIARES.SEMPRE_1 AND "DB GRUPO 1".STAT48.STAT92;
   "Q207" := "DB PRINCIPAL".AUXILIARES.SEMPRE_1 AND "DB GRUPO 1".STAT48.STAT93;
   "Q210" := "DB PRINCIPAL".AUXILIARES.SEMPRE_1 AND "DB GRUPO 1".STAT48.STAT94;
END_REGION

REGION Network 17: LIBERA GAS QUEIMADORES
   RUNG wire#powerrail
      Contact( "DB PRINCIPAL".AUXILIARES.SEMPRE_1 )
      wire#w1
      Contact( "I210" )
      wire#w2
      Coil( "Q203" )
   END_RUNG
   RUNG wire#w1
      Contact( "I212" )
   END_RUNG wire#w2
   RUNG wire#w2
      Coil( "DB GRUPO 1".STAT96.STAT133 )
   END_RUNG
   RUNG wire#w1
      Contact( "I211" )
      wire#w3
      Coil( "Q202" )
   END_RUNG
   RUNG wire#w1
      Contact( "I213" )
   END_RUNG wire#w3
   RUNG wire#w1
      Contact( %DB2.DBX13.7 )
   END_RUNG wire#w3
   RUNG wire#w3
      Coil( "DB GRUPO 1".STAT96.STAT134 )
   END_RUNG
   // the same network as SCL:
   "Q203" := "DB PRINCIPAL".AUXILIARES.SEMPRE_1 AND ("I210" OR "I212");
   "DB GRUPO 1".STAT96.STAT133 := "Q203";
   "Q202" := "DB PRINCIPAL".AUXILIARES.SEMPRE_1 AND ("I211" OR "I213" OR %DB2.DBX13.7);
   "DB GRUPO 1".STAT96.STAT134 := "Q202";
END_REGION

REGION Network 18: ESCOVAS 1 E 2
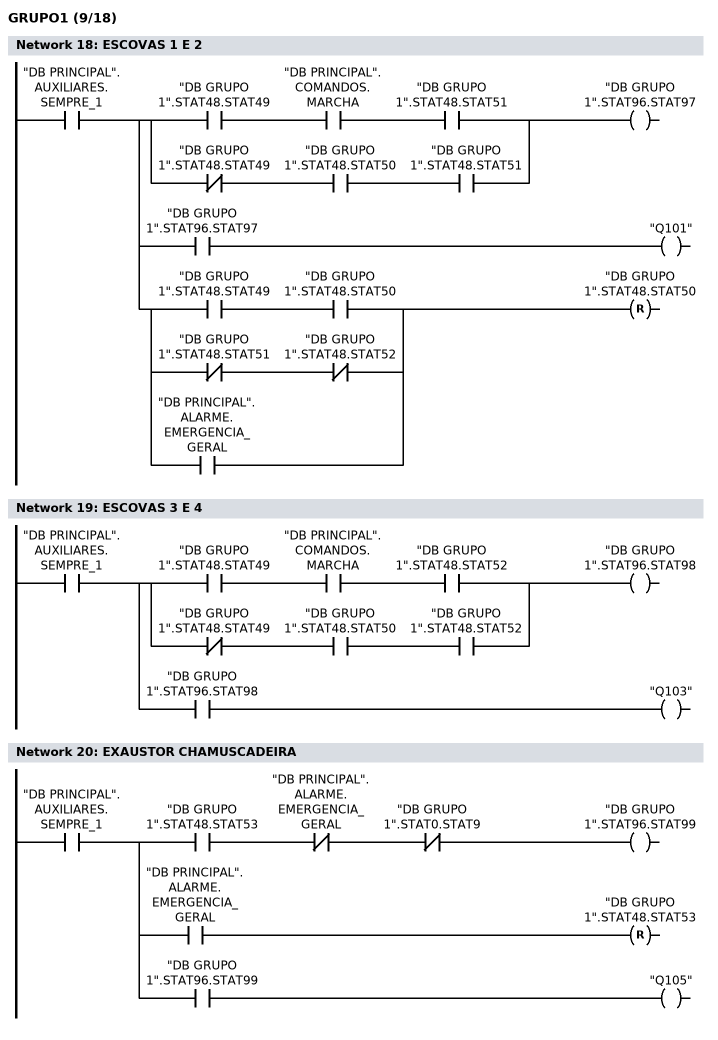
   RUNG wire#powerrail
      Contact( "DB PRINCIPAL".AUXILIARES.SEMPRE_1 )
      wire#w1
      Contact( "DB GRUPO 1".STAT48.STAT49 )
      Contact( "DB PRINCIPAL".COMANDOS.MARCHA )
      Contact( "DB GRUPO 1".STAT48.STAT51 )
      wire#w2
      Coil( "DB GRUPO 1".STAT96.STAT97 )
   END_RUNG
   RUNG wire#w1
      I_Contact( "DB GRUPO 1".STAT48.STAT49 )
      Contact( "DB GRUPO 1".STAT48.STAT50 )
      Contact( "DB GRUPO 1".STAT48.STAT51 )
   END_RUNG wire#w2
   RUNG wire#w1
      Contact( "DB GRUPO 1".STAT96.STAT97 )
      Coil( "Q101" )
   END_RUNG
   RUNG wire#w1
      Contact( "DB GRUPO 1".STAT48.STAT49 )
      Contact( "DB GRUPO 1".STAT48.STAT50 )
      wire#w3
      R_Coil( "DB GRUPO 1".STAT48.STAT50 )
   END_RUNG
   RUNG wire#w1
      I_Contact( "DB GRUPO 1".STAT48.STAT51 )
      I_Contact( "DB GRUPO 1".STAT48.STAT52 )
   END_RUNG wire#w3
   RUNG wire#w1
      Contact( "DB PRINCIPAL".ALARME.EMERGENCIA_GERAL )
   END_RUNG wire#w3
   // the same network as SCL:
   "DB GRUPO 1".STAT96.STAT97 := "DB PRINCIPAL".AUXILIARES.SEMPRE_1 AND (("DB GRUPO 1".STAT48.STAT49 AND "DB PRINCIPAL".COMANDOS.MARCHA AND "DB GRUPO 1".STAT48.STAT51) OR (NOT "DB GRUPO 1".STAT48.STAT49 AND "DB GRUPO 1".STAT48.STAT50 AND "DB GRUPO 1".STAT48.STAT51));
   "Q101" := "DB PRINCIPAL".AUXILIARES.SEMPRE_1 AND "DB GRUPO 1".STAT96.STAT97;
   IF "DB PRINCIPAL".AUXILIARES.SEMPRE_1 AND (("DB GRUPO 1".STAT48.STAT49 AND "DB GRUPO 1".STAT48.STAT50) OR (NOT "DB GRUPO 1".STAT48.STAT51 AND NOT "DB GRUPO 1".STAT48.STAT52) OR "DB PRINCIPAL".ALARME.EMERGENCIA_GERAL) THEN
       "DB GRUPO 1".STAT48.STAT50 := FALSE;
   END_IF;
END_REGION

REGION Network 19: ESCOVAS 3 E 4
   RUNG wire#powerrail
      Contact( "DB PRINCIPAL".AUXILIARES.SEMPRE_1 )
      wire#w1
      Contact( "DB GRUPO 1".STAT48.STAT49 )
      Contact( "DB PRINCIPAL".COMANDOS.MARCHA )
      Contact( "DB GRUPO 1".STAT48.STAT52 )
      wire#w2
      Coil( "DB GRUPO 1".STAT96.STAT98 )
   END_RUNG
   RUNG wire#w1
      I_Contact( "DB GRUPO 1".STAT48.STAT49 )
      Contact( "DB GRUPO 1".STAT48.STAT50 )
      Contact( "DB GRUPO 1".STAT48.STAT52 )
   END_RUNG wire#w2
   RUNG wire#w1
      Contact( "DB GRUPO 1".STAT96.STAT98 )
      Coil( "Q103" )
   END_RUNG
   // the same network as SCL:
   "DB GRUPO 1".STAT96.STAT98 := "DB PRINCIPAL".AUXILIARES.SEMPRE_1 AND (("DB GRUPO 1".STAT48.STAT49 AND "DB PRINCIPAL".COMANDOS.MARCHA AND "DB GRUPO 1".STAT48.STAT52) OR (NOT "DB GRUPO 1".STAT48.STAT49 AND "DB GRUPO 1".STAT48.STAT50 AND "DB GRUPO 1".STAT48.STAT52));
   "Q103" := "DB PRINCIPAL".AUXILIARES.SEMPRE_1 AND "DB GRUPO 1".STAT96.STAT98;
END_REGION

REGION Network 20: EXAUSTOR CHAMUSCADEIRA
   RUNG wire#powerrail
      Contact( "DB PRINCIPAL".AUXILIARES.SEMPRE_1 )
      wire#w1
      Contact( "DB GRUPO 1".STAT48.STAT53 )
      I_Contact( "DB PRINCIPAL".ALARME.EMERGENCIA_GERAL )
      I_Contact( "DB GRUPO 1".STAT0.STAT9 )
      Coil( "DB GRUPO 1".STAT96.STAT99 )
   END_RUNG
   RUNG wire#w1
      Contact( "DB PRINCIPAL".ALARME.EMERGENCIA_GERAL )
      R_Coil( "DB GRUPO 1".STAT48.STAT53 )
   END_RUNG
   RUNG wire#w1
      Contact( "DB GRUPO 1".STAT96.STAT99 )
      Coil( "Q105" )
   END_RUNG
   // the same network as SCL:
   "DB GRUPO 1".STAT96.STAT99 := "DB PRINCIPAL".AUXILIARES.SEMPRE_1 AND "DB GRUPO 1".STAT48.STAT53 AND NOT "DB PRINCIPAL".ALARME.EMERGENCIA_GERAL AND NOT "DB GRUPO 1".STAT0.STAT9;
   IF "DB PRINCIPAL".AUXILIARES.SEMPRE_1 AND "DB PRINCIPAL".ALARME.EMERGENCIA_GERAL THEN
       "DB GRUPO 1".STAT48.STAT53 := FALSE;
   END_IF;
   "Q105" := "DB PRINCIPAL".AUXILIARES.SEMPRE_1 AND "DB GRUPO 1".STAT96.STAT99;
END_REGION

REGION Network 21: VENTILADOR 1 CHAMUSCADEIRA
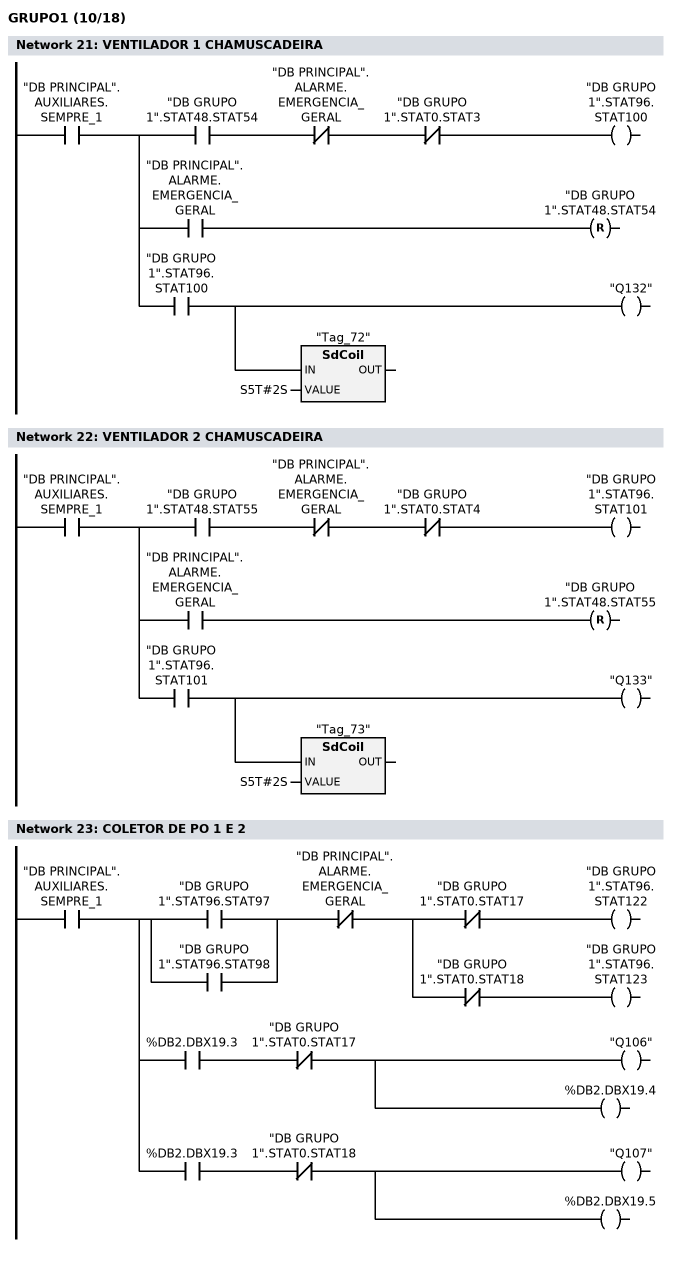
   // no SCL statement known for SdCoil: written as a call
   "DB GRUPO 1".STAT96.STAT100 := "DB PRINCIPAL".AUXILIARES.SEMPRE_1 AND "DB GRUPO 1".STAT48.STAT54 AND NOT "DB PRINCIPAL".ALARME.EMERGENCIA_GERAL AND NOT "DB GRUPO 1".STAT0.STAT3;
   IF "DB PRINCIPAL".AUXILIARES.SEMPRE_1 AND "DB PRINCIPAL".ALARME.EMERGENCIA_GERAL THEN
       "DB GRUPO 1".STAT48.STAT54 := FALSE;
   END_IF;
   "Q132" := "DB PRINCIPAL".AUXILIARES.SEMPRE_1 AND "DB GRUPO 1".STAT96.STAT100;
   SdCoil(value := S5T#2S, operand := "Tag_72", in := "Q132");
END_REGION

REGION Network 22: VENTILADOR 2 CHAMUSCADEIRA
   // no SCL statement known for SdCoil: written as a call
   "DB GRUPO 1".STAT96.STAT101 := "DB PRINCIPAL".AUXILIARES.SEMPRE_1 AND "DB GRUPO 1".STAT48.STAT55 AND NOT "DB PRINCIPAL".ALARME.EMERGENCIA_GERAL AND NOT "DB GRUPO 1".STAT0.STAT4;
   IF "DB PRINCIPAL".AUXILIARES.SEMPRE_1 AND "DB PRINCIPAL".ALARME.EMERGENCIA_GERAL THEN
       "DB GRUPO 1".STAT48.STAT55 := FALSE;
   END_IF;
   "Q133" := "DB PRINCIPAL".AUXILIARES.SEMPRE_1 AND "DB GRUPO 1".STAT96.STAT101;
   SdCoil(value := S5T#2S, operand := "Tag_73", in := "Q133");
END_REGION

REGION Network 23: COLETOR DE PO 1 E 2
   RUNG wire#powerrail
      Contact( "DB PRINCIPAL".AUXILIARES.SEMPRE_1 )
      wire#w1
      Contact( "DB GRUPO 1".STAT96.STAT97 )
      wire#w2
      I_Contact( "DB PRINCIPAL".ALARME.EMERGENCIA_GERAL )
      wire#w3
      I_Contact( "DB GRUPO 1".STAT0.STAT17 )
      Coil( "DB GRUPO 1".STAT96.STAT122 )
   END_RUNG
   RUNG wire#w1
      Contact( "DB GRUPO 1".STAT96.STAT98 )
   END_RUNG wire#w2
   RUNG wire#w3
      I_Contact( "DB GRUPO 1".STAT0.STAT18 )
      Coil( "DB GRUPO 1".STAT96.STAT123 )
   END_RUNG
   RUNG wire#w1
      Contact( %DB2.DBX19.3 )
      I_Contact( "DB GRUPO 1".STAT0.STAT17 )
      wire#w4
      Coil( "Q106" )
   END_RUNG
   RUNG wire#w4
      Coil( %DB2.DBX19.4 )
   END_RUNG
   RUNG wire#w1
      Contact( %DB2.DBX19.3 )
      I_Contact( "DB GRUPO 1".STAT0.STAT18 )
      wire#w5
      Coil( "Q107" )
   END_RUNG
   RUNG wire#w5
      Coil( %DB2.DBX19.5 )
   END_RUNG
   // the same network as SCL:
   #_w1 := "DB PRINCIPAL".AUXILIARES.SEMPRE_1 AND ("DB GRUPO 1".STAT96.STAT97 OR "DB GRUPO 1".STAT96.STAT98) AND NOT "DB PRINCIPAL".ALARME.EMERGENCIA_GERAL;
   "DB GRUPO 1".STAT96.STAT122 := #_w1 AND NOT "DB GRUPO 1".STAT0.STAT17;
   "DB GRUPO 1".STAT96.STAT123 := #_w1 AND NOT "DB GRUPO 1".STAT0.STAT18;
   "Q106" := "DB PRINCIPAL".AUXILIARES.SEMPRE_1 AND %DB2.DBX19.3 AND NOT "DB GRUPO 1".STAT0.STAT17;
   %DB2.DBX19.4 := "Q106";
   "Q107" := "DB PRINCIPAL".AUXILIARES.SEMPRE_1 AND %DB2.DBX19.3 AND NOT "DB GRUPO 1".STAT0.STAT18;
   %DB2.DBX19.5 := "Q107";
END_REGION

REGION Network 24: EXAUSTOR NEUTRALIZAÇÃO 1
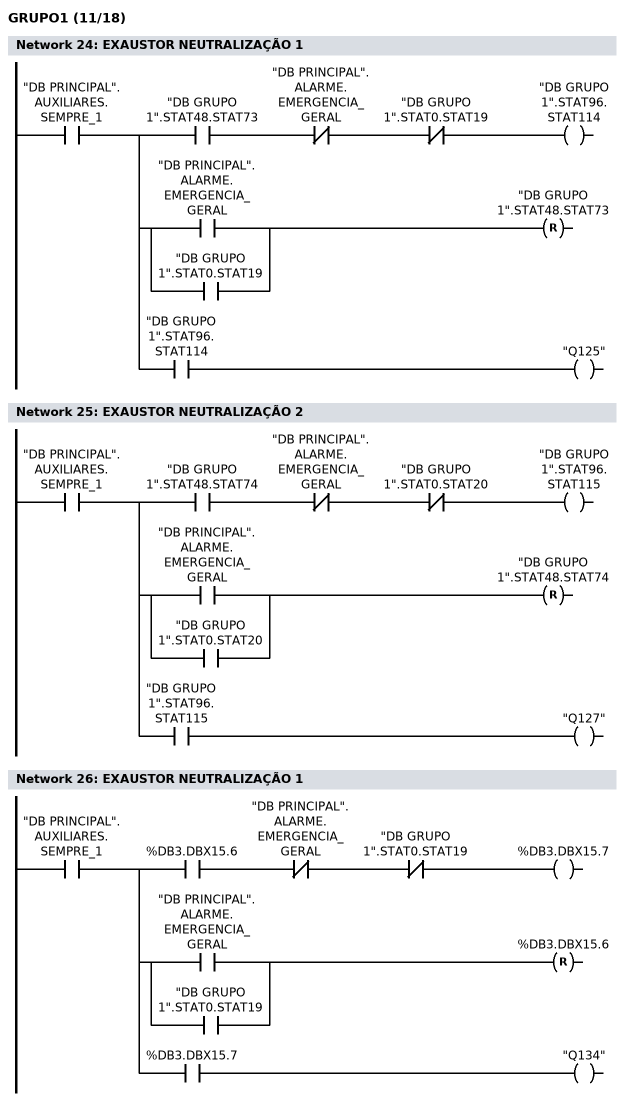
   RUNG wire#powerrail
      Contact( "DB PRINCIPAL".AUXILIARES.SEMPRE_1 )
      wire#w1
      Contact( "DB GRUPO 1".STAT48.STAT73 )
      I_Contact( "DB PRINCIPAL".ALARME.EMERGENCIA_GERAL )
      I_Contact( "DB GRUPO 1".STAT0.STAT19 )
      Coil( "DB GRUPO 1".STAT96.STAT114 )
   END_RUNG
   RUNG wire#w1
      Contact( "DB PRINCIPAL".ALARME.EMERGENCIA_GERAL )
      wire#w2
      R_Coil( "DB GRUPO 1".STAT48.STAT73 )
   END_RUNG
   RUNG wire#w1
      Contact( "DB GRUPO 1".STAT0.STAT19 )
   END_RUNG wire#w2
   RUNG wire#w1
      Contact( "DB GRUPO 1".STAT96.STAT114 )
      Coil( "Q125" )
   END_RUNG
   // the same network as SCL:
   "DB GRUPO 1".STAT96.STAT114 := "DB PRINCIPAL".AUXILIARES.SEMPRE_1 AND "DB GRUPO 1".STAT48.STAT73 AND NOT "DB PRINCIPAL".ALARME.EMERGENCIA_GERAL AND NOT "DB GRUPO 1".STAT0.STAT19;
   IF "DB PRINCIPAL".AUXILIARES.SEMPRE_1 AND ("DB PRINCIPAL".ALARME.EMERGENCIA_GERAL OR "DB GRUPO 1".STAT0.STAT19) THEN
       "DB GRUPO 1".STAT48.STAT73 := FALSE;
   END_IF;
   "Q125" := "DB PRINCIPAL".AUXILIARES.SEMPRE_1 AND "DB GRUPO 1".STAT96.STAT114;
END_REGION

REGION Network 25: EXAUSTOR NEUTRALIZAÇÃO 2
   RUNG wire#powerrail
      Contact( "DB PRINCIPAL".AUXILIARES.SEMPRE_1 )
      wire#w1
      Contact( "DB GRUPO 1".STAT48.STAT74 )
      I_Contact( "DB PRINCIPAL".ALARME.EMERGENCIA_GERAL )
      I_Contact( "DB GRUPO 1".STAT0.STAT20 )
      Coil( "DB GRUPO 1".STAT96.STAT115 )
   END_RUNG
   RUNG wire#w1
      Contact( "DB PRINCIPAL".ALARME.EMERGENCIA_GERAL )
      wire#w2
      R_Coil( "DB GRUPO 1".STAT48.STAT74 )
   END_RUNG
   RUNG wire#w1
      Contact( "DB GRUPO 1".STAT0.STAT20 )
   END_RUNG wire#w2
   RUNG wire#w1
      Contact( "DB GRUPO 1".STAT96.STAT115 )
      Coil( "Q127" )
   END_RUNG
   // the same network as SCL:
   "DB GRUPO 1".STAT96.STAT115 := "DB PRINCIPAL".AUXILIARES.SEMPRE_1 AND "DB GRUPO 1".STAT48.STAT74 AND NOT "DB PRINCIPAL".ALARME.EMERGENCIA_GERAL AND NOT "DB GRUPO 1".STAT0.STAT20;
   IF "DB PRINCIPAL".AUXILIARES.SEMPRE_1 AND ("DB PRINCIPAL".ALARME.EMERGENCIA_GERAL OR "DB GRUPO 1".STAT0.STAT20) THEN
       "DB GRUPO 1".STAT48.STAT74 := FALSE;
   END_IF;
   "Q127" := "DB PRINCIPAL".AUXILIARES.SEMPRE_1 AND "DB GRUPO 1".STAT96.STAT115;
END_REGION

REGION Network 26: EXAUSTOR NEUTRALIZAÇÃO 1
   RUNG wire#powerrail
      Contact( "DB PRINCIPAL".AUXILIARES.SEMPRE_1 )
      wire#w1
      Contact( %DB3.DBX15.6 )
      I_Contact( "DB PRINCIPAL".ALARME.EMERGENCIA_GERAL )
      I_Contact( "DB GRUPO 1".STAT0.STAT19 )
      Coil( %DB3.DBX15.7 )
   END_RUNG
   RUNG wire#w1
      Contact( "DB PRINCIPAL".ALARME.EMERGENCIA_GERAL )
      wire#w2
      R_Coil( %DB3.DBX15.6 )
   END_RUNG
   RUNG wire#w1
      Contact( "DB GRUPO 1".STAT0.STAT19 )
   END_RUNG wire#w2
   RUNG wire#w1
      Contact( %DB3.DBX15.7 )
      Coil( "Q134" )
   END_RUNG
   // the same network as SCL:
   %DB3.DBX15.7 := "DB PRINCIPAL".AUXILIARES.SEMPRE_1 AND %DB3.DBX15.6 AND NOT "DB PRINCIPAL".ALARME.EMERGENCIA_GERAL AND NOT "DB GRUPO 1".STAT0.STAT19;
   IF "DB PRINCIPAL".AUXILIARES.SEMPRE_1 AND ("DB PRINCIPAL".ALARME.EMERGENCIA_GERAL OR "DB GRUPO 1".STAT0.STAT19) THEN
       %DB3.DBX15.6 := FALSE;
   END_IF;
   "Q134" := "DB PRINCIPAL".AUXILIARES.SEMPRE_1 AND %DB3.DBX15.7;
END_REGION

REGION Network 27: BOMBA DE CIRCULAÇÃO NEUTRALIZAÇÃO 1
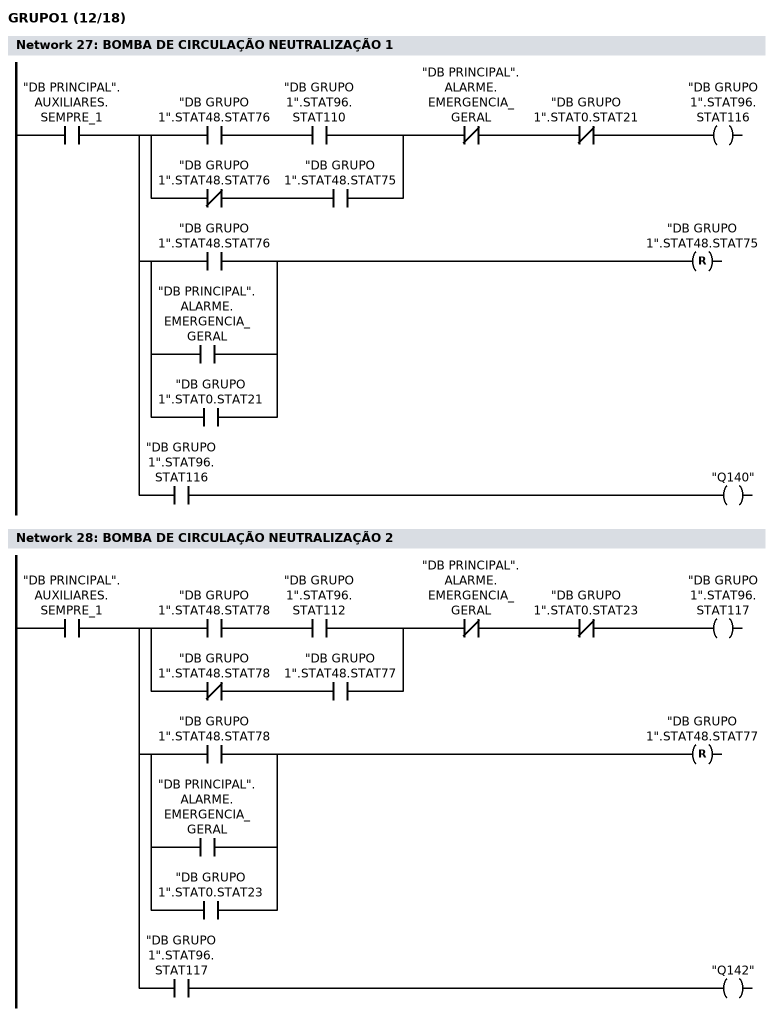
   RUNG wire#powerrail
      Contact( "DB PRINCIPAL".AUXILIARES.SEMPRE_1 )
      wire#w1
      Contact( "DB GRUPO 1".STAT48.STAT76 )
      Contact( "DB GRUPO 1".STAT96.STAT110 )
      wire#w2
      I_Contact( "DB PRINCIPAL".ALARME.EMERGENCIA_GERAL )
      I_Contact( "DB GRUPO 1".STAT0.STAT21 )
      Coil( "DB GRUPO 1".STAT96.STAT116 )
   END_RUNG
   RUNG wire#w1
      I_Contact( "DB GRUPO 1".STAT48.STAT76 )
      Contact( "DB GRUPO 1".STAT48.STAT75 )
   END_RUNG wire#w2
   RUNG wire#w1
      Contact( "DB GRUPO 1".STAT48.STAT76 )
      wire#w3
      R_Coil( "DB GRUPO 1".STAT48.STAT75 )
   END_RUNG
   RUNG wire#w1
      Contact( "DB PRINCIPAL".ALARME.EMERGENCIA_GERAL )
   END_RUNG wire#w3
   RUNG wire#w1
      Contact( "DB GRUPO 1".STAT0.STAT21 )
   END_RUNG wire#w3
   RUNG wire#w1
      Contact( "DB GRUPO 1".STAT96.STAT116 )
      Coil( "Q140" )
   END_RUNG
   // the same network as SCL:
   "DB GRUPO 1".STAT96.STAT116 := "DB PRINCIPAL".AUXILIARES.SEMPRE_1 AND (("DB GRUPO 1".STAT48.STAT76 AND "DB GRUPO 1".STAT96.STAT110) OR (NOT "DB GRUPO 1".STAT48.STAT76 AND "DB GRUPO 1".STAT48.STAT75)) AND NOT "DB PRINCIPAL".ALARME.EMERGENCIA_GERAL AND NOT "DB GRUPO 1".STAT0.STAT21;
   IF "DB PRINCIPAL".AUXILIARES.SEMPRE_1 AND ("DB GRUPO 1".STAT48.STAT76 OR "DB PRINCIPAL".ALARME.EMERGENCIA_GERAL OR "DB GRUPO 1".STAT0.STAT21) THEN
       "DB GRUPO 1".STAT48.STAT75 := FALSE;
   END_IF;
   "Q140" := "DB PRINCIPAL".AUXILIARES.SEMPRE_1 AND "DB GRUPO 1".STAT96.STAT116;
END_REGION

REGION Network 28: BOMBA DE CIRCULAÇÃO NEUTRALIZAÇÃO 2
   RUNG wire#powerrail
      Contact( "DB PRINCIPAL".AUXILIARES.SEMPRE_1 )
      wire#w1
      Contact( "DB GRUPO 1".STAT48.STAT78 )
      Contact( "DB GRUPO 1".STAT96.STAT112 )
      wire#w2
      I_Contact( "DB PRINCIPAL".ALARME.EMERGENCIA_GERAL )
      I_Contact( "DB GRUPO 1".STAT0.STAT23 )
      Coil( "DB GRUPO 1".STAT96.STAT117 )
   END_RUNG
   RUNG wire#w1
      I_Contact( "DB GRUPO 1".STAT48.STAT78 )
      Contact( "DB GRUPO 1".STAT48.STAT77 )
   END_RUNG wire#w2
   RUNG wire#w1
      Contact( "DB GRUPO 1".STAT48.STAT78 )
      wire#w3
      R_Coil( "DB GRUPO 1".STAT48.STAT77 )
   END_RUNG
   RUNG wire#w1
      Contact( "DB PRINCIPAL".ALARME.EMERGENCIA_GERAL )
   END_RUNG wire#w3
   RUNG wire#w1
      Contact( "DB GRUPO 1".STAT0.STAT23 )
   END_RUNG wire#w3
   RUNG wire#w1
      Contact( "DB GRUPO 1".STAT96.STAT117 )
      Coil( "Q142" )
   END_RUNG
   // the same network as SCL:
   "DB GRUPO 1".STAT96.STAT117 := "DB PRINCIPAL".AUXILIARES.SEMPRE_1 AND (("DB GRUPO 1".STAT48.STAT78 AND "DB GRUPO 1".STAT96.STAT112) OR (NOT "DB GRUPO 1".STAT48.STAT78 AND "DB GRUPO 1".STAT48.STAT77)) AND NOT "DB PRINCIPAL".ALARME.EMERGENCIA_GERAL AND NOT "DB GRUPO 1".STAT0.STAT23;
   IF "DB PRINCIPAL".AUXILIARES.SEMPRE_1 AND ("DB GRUPO 1".STAT48.STAT78 OR "DB PRINCIPAL".ALARME.EMERGENCIA_GERAL OR "DB GRUPO 1".STAT0.STAT23) THEN
       "DB GRUPO 1".STAT48.STAT77 := FALSE;
   END_IF;
   "Q142" := "DB PRINCIPAL".AUXILIARES.SEMPRE_1 AND "DB GRUPO 1".STAT96.STAT117;
END_REGION

REGION Network 29: FILTRO ROTATIVO NEUTRALIZAÇÃO 1
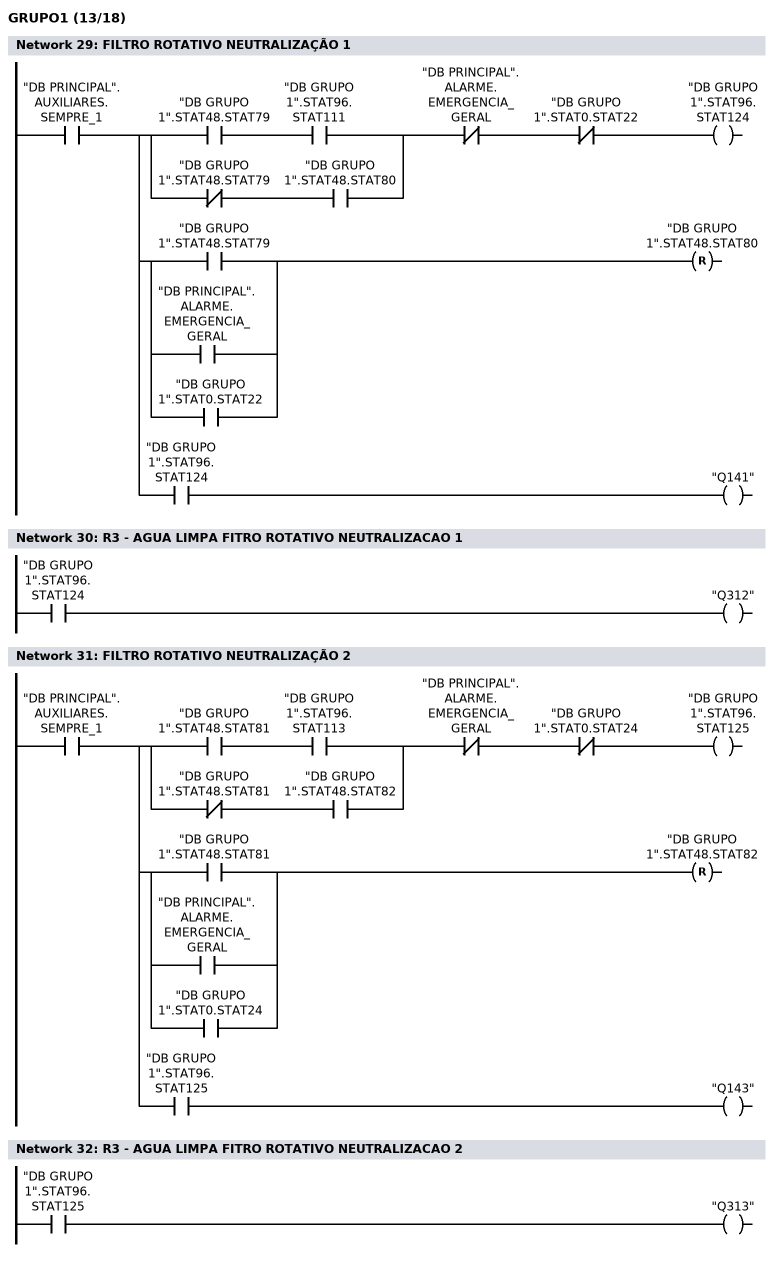
   RUNG wire#powerrail
      Contact( "DB PRINCIPAL".AUXILIARES.SEMPRE_1 )
      wire#w1
      Contact( "DB GRUPO 1".STAT48.STAT79 )
      Contact( "DB GRUPO 1".STAT96.STAT111 )
      wire#w2
      I_Contact( "DB PRINCIPAL".ALARME.EMERGENCIA_GERAL )
      I_Contact( "DB GRUPO 1".STAT0.STAT22 )
      Coil( "DB GRUPO 1".STAT96.STAT124 )
   END_RUNG
   RUNG wire#w1
      I_Contact( "DB GRUPO 1".STAT48.STAT79 )
      Contact( "DB GRUPO 1".STAT48.STAT80 )
   END_RUNG wire#w2
   RUNG wire#w1
      Contact( "DB GRUPO 1".STAT48.STAT79 )
      wire#w3
      R_Coil( "DB GRUPO 1".STAT48.STAT80 )
   END_RUNG
   RUNG wire#w1
      Contact( "DB PRINCIPAL".ALARME.EMERGENCIA_GERAL )
   END_RUNG wire#w3
   RUNG wire#w1
      Contact( "DB GRUPO 1".STAT0.STAT22 )
   END_RUNG wire#w3
   RUNG wire#w1
      Contact( "DB GRUPO 1".STAT96.STAT124 )
      Coil( "Q141" )
   END_RUNG
   // the same network as SCL:
   "DB GRUPO 1".STAT96.STAT124 := "DB PRINCIPAL".AUXILIARES.SEMPRE_1 AND (("DB GRUPO 1".STAT48.STAT79 AND "DB GRUPO 1".STAT96.STAT111) OR (NOT "DB GRUPO 1".STAT48.STAT79 AND "DB GRUPO 1".STAT48.STAT80)) AND NOT "DB PRINCIPAL".ALARME.EMERGENCIA_GERAL AND NOT "DB GRUPO 1".STAT0.STAT22;
   IF "DB PRINCIPAL".AUXILIARES.SEMPRE_1 AND ("DB GRUPO 1".STAT48.STAT79 OR "DB PRINCIPAL".ALARME.EMERGENCIA_GERAL OR "DB GRUPO 1".STAT0.STAT22) THEN
       "DB GRUPO 1".STAT48.STAT80 := FALSE;
   END_IF;
   "Q141" := "DB PRINCIPAL".AUXILIARES.SEMPRE_1 AND "DB GRUPO 1".STAT96.STAT124;
END_REGION

REGION Network 30: R3 - AGUA LIMPA FITRO ROTATIVO NEUTRALIZACAO 1
   RUNG wire#powerrail
      Contact( "DB GRUPO 1".STAT96.STAT124 )
      Coil( "Q312" )
   END_RUNG
   // the same network as SCL:
   "Q312" := "DB GRUPO 1".STAT96.STAT124;
END_REGION

REGION Network 31: FILTRO ROTATIVO NEUTRALIZAÇÃO 2
   RUNG wire#powerrail
      Contact( "DB PRINCIPAL".AUXILIARES.SEMPRE_1 )
      wire#w1
      Contact( "DB GRUPO 1".STAT48.STAT81 )
      Contact( "DB GRUPO 1".STAT96.STAT113 )
      wire#w2
      I_Contact( "DB PRINCIPAL".ALARME.EMERGENCIA_GERAL )
      I_Contact( "DB GRUPO 1".STAT0.STAT24 )
      Coil( "DB GRUPO 1".STAT96.STAT125 )
   END_RUNG
   RUNG wire#w1
      I_Contact( "DB GRUPO 1".STAT48.STAT81 )
      Contact( "DB GRUPO 1".STAT48.STAT82 )
   END_RUNG wire#w2
   RUNG wire#w1
      Contact( "DB GRUPO 1".STAT48.STAT81 )
      wire#w3
      R_Coil( "DB GRUPO 1".STAT48.STAT82 )
   END_RUNG
   RUNG wire#w1
      Contact( "DB PRINCIPAL".ALARME.EMERGENCIA_GERAL )
   END_RUNG wire#w3
   RUNG wire#w1
      Contact( "DB GRUPO 1".STAT0.STAT24 )
   END_RUNG wire#w3
   RUNG wire#w1
      Contact( "DB GRUPO 1".STAT96.STAT125 )
      Coil( "Q143" )
   END_RUNG
   // the same network as SCL:
   "DB GRUPO 1".STAT96.STAT125 := "DB PRINCIPAL".AUXILIARES.SEMPRE_1 AND (("DB GRUPO 1".STAT48.STAT81 AND "DB GRUPO 1".STAT96.STAT113) OR (NOT "DB GRUPO 1".STAT48.STAT81 AND "DB GRUPO 1".STAT48.STAT82)) AND NOT "DB PRINCIPAL".ALARME.EMERGENCIA_GERAL AND NOT "DB GRUPO 1".STAT0.STAT24;
   IF "DB PRINCIPAL".AUXILIARES.SEMPRE_1 AND ("DB GRUPO 1".STAT48.STAT81 OR "DB PRINCIPAL".ALARME.EMERGENCIA_GERAL OR "DB GRUPO 1".STAT0.STAT24) THEN
       "DB GRUPO 1".STAT48.STAT82 := FALSE;
   END_IF;
   "Q143" := "DB PRINCIPAL".AUXILIARES.SEMPRE_1 AND "DB GRUPO 1".STAT96.STAT125;
END_REGION

REGION Network 32: R3 - AGUA LIMPA FITRO ROTATIVO NEUTRALIZACAO 2
   RUNG wire#powerrail
      Contact( "DB GRUPO 1".STAT96.STAT125 )
      Coil( "Q313" )
   END_RUNG
   // the same network as SCL:
   "Q313" := "DB GRUPO 1".STAT96.STAT125;
END_REGION

REGION Network 33: NIVEIS NEUTRALIZACAO 1
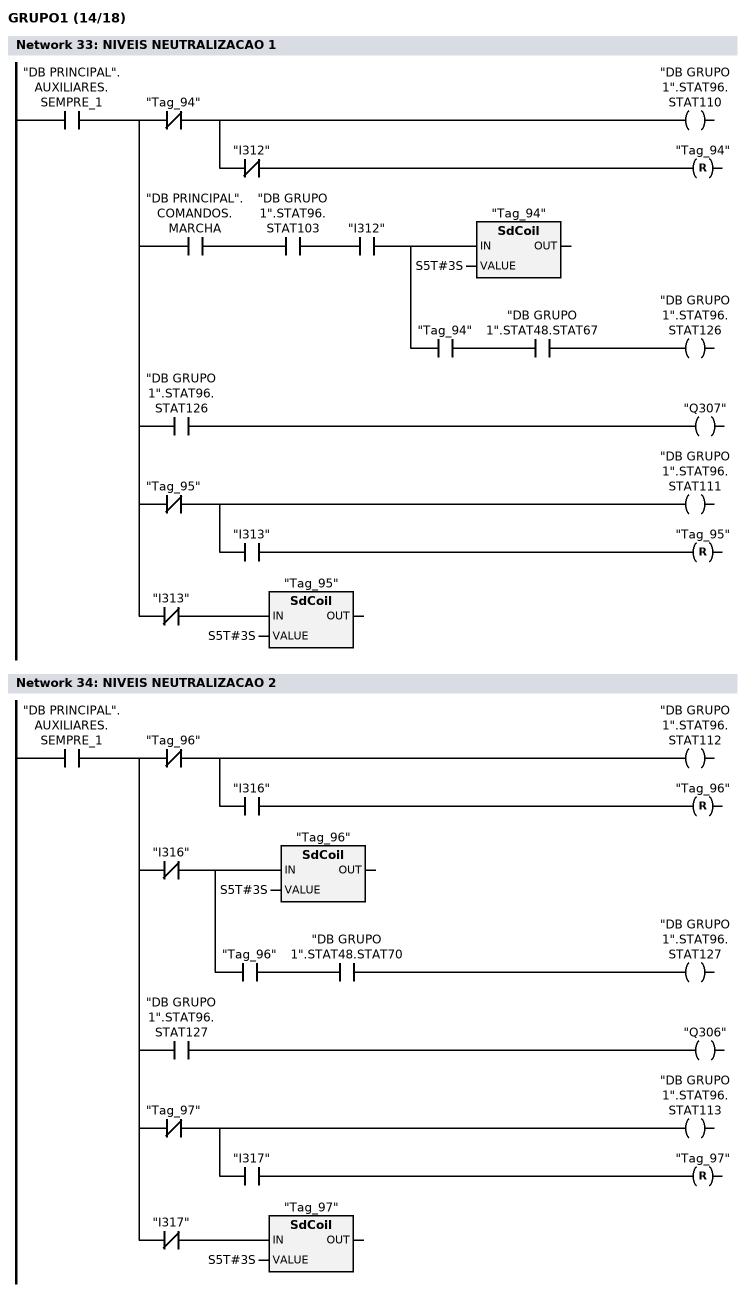
   // no SCL statement known for SdCoil: written as a call
   "DB GRUPO 1".STAT96.STAT110 := "DB PRINCIPAL".AUXILIARES.SEMPRE_1 AND NOT "Tag_94";
   IF "DB GRUPO 1".STAT96.STAT110 AND NOT "I312" THEN "Tag_94" := FALSE; END_IF;
   #_w1 := "DB PRINCIPAL".AUXILIARES.SEMPRE_1 AND "DB PRINCIPAL".COMANDOS.MARCHA AND "DB GRUPO 1".STAT96.STAT103 AND "I312";
   #_w2 := "DB PRINCIPAL".AUXILIARES.SEMPRE_1;
   SdCoil(value := S5T#3S, operand := "Tag_94", in := #_w1);
   "DB GRUPO 1".STAT96.STAT126 := #_w1 AND "Tag_94" AND "DB GRUPO 1".STAT48.STAT67;
   "Q307" := #_w2 AND "DB GRUPO 1".STAT96.STAT126;
   "DB GRUPO 1".STAT96.STAT111 := #_w2 AND NOT "Tag_95";
   IF "DB GRUPO 1".STAT96.STAT111 AND "I313" THEN "Tag_95" := FALSE; END_IF;
   SdCoil(value := S5T#3S, operand := "Tag_95", in := #_w2 AND NOT "I313");
END_REGION

REGION Network 34: NIVEIS NEUTRALIZACAO 2
   // no SCL statement known for SdCoil: written as a call
   "DB GRUPO 1".STAT96.STAT112 := "DB PRINCIPAL".AUXILIARES.SEMPRE_1 AND NOT "Tag_96";
   IF "DB GRUPO 1".STAT96.STAT112 AND "I316" THEN "Tag_96" := FALSE; END_IF;
   #_w1 := "DB PRINCIPAL".AUXILIARES.SEMPRE_1 AND NOT "I316";
   #_w2 := "DB PRINCIPAL".AUXILIARES.SEMPRE_1;
   SdCoil(value := S5T#3S, operand := "Tag_96", in := #_w1);
   "DB GRUPO 1".STAT96.STAT127 := #_w1 AND "Tag_96" AND "DB GRUPO 1".STAT48.STAT70;
   "Q306" := #_w2 AND "DB GRUPO 1".STAT96.STAT127;
   "DB GRUPO 1".STAT96.STAT113 := #_w2 AND NOT "Tag_97";
   IF "DB GRUPO 1".STAT96.STAT113 AND "I317" THEN "Tag_97" := FALSE; END_IF;
   SdCoil(value := S5T#3S, operand := "Tag_97", in := #_w2 AND NOT "I317");
END_REGION

REGION Network 35: BOMBA 3 CIRCULAÇÃO DA LAVAGEM
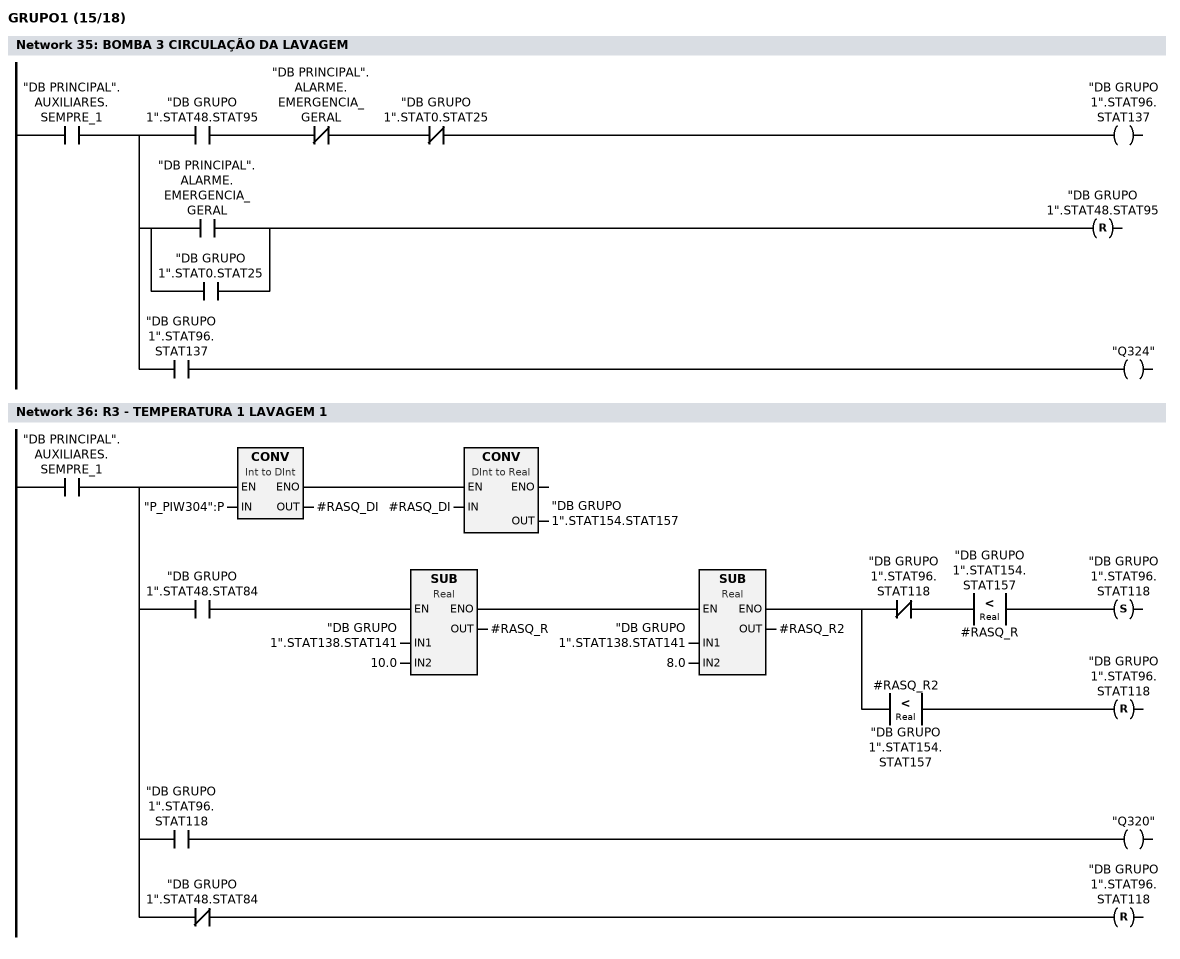
   RUNG wire#powerrail
      Contact( "DB PRINCIPAL".AUXILIARES.SEMPRE_1 )
      wire#w1
      Contact( "DB GRUPO 1".STAT48.STAT95 )
      I_Contact( "DB PRINCIPAL".ALARME.EMERGENCIA_GERAL )
      I_Contact( "DB GRUPO 1".STAT0.STAT25 )
      Coil( "DB GRUPO 1".STAT96.STAT137 )
   END_RUNG
   RUNG wire#w1
      Contact( "DB PRINCIPAL".ALARME.EMERGENCIA_GERAL )
      wire#w2
      R_Coil( "DB GRUPO 1".STAT48.STAT95 )
   END_RUNG
   RUNG wire#w1
      Contact( "DB GRUPO 1".STAT0.STAT25 )
   END_RUNG wire#w2
   RUNG wire#w1
      Contact( "DB GRUPO 1".STAT96.STAT137 )
      Coil( "Q324" )
   END_RUNG
   // the same network as SCL:
   "DB GRUPO 1".STAT96.STAT137 := "DB PRINCIPAL".AUXILIARES.SEMPRE_1 AND "DB GRUPO 1".STAT48.STAT95 AND NOT "DB PRINCIPAL".ALARME.EMERGENCIA_GERAL AND NOT "DB GRUPO 1".STAT0.STAT25;
   IF "DB PRINCIPAL".AUXILIARES.SEMPRE_1 AND ("DB PRINCIPAL".ALARME.EMERGENCIA_GERAL OR "DB GRUPO 1".STAT0.STAT25) THEN
       "DB GRUPO 1".STAT48.STAT95 := FALSE;
   END_IF;
   "Q324" := "DB PRINCIPAL".AUXILIARES.SEMPRE_1 AND "DB GRUPO 1".STAT96.STAT137;
END_REGION

REGION Network 36: R3 - TEMPERATURA 1 LAVAGEM 1
   RUNG wire#powerrail
      Contact( "DB PRINCIPAL".AUXILIARES.SEMPRE_1 )
      wire#w1
      { S7_Templates := "[SrcType := Int, DestType := DInt]"; S7_GenerateENO := "TRUE" } Convert(in := "P_PIW304":P, out => #RASQ_DI)
      { S7_Templates := "[SrcType := DInt, DestType := Real]"; S7_GenerateENO := "TRUE" } Convert(in := #RASQ_DI, out => "DB GRUPO 1".STAT154.STAT157)
   END_RUNG
   RUNG wire#w1
      Contact( "DB GRUPO 1".STAT48.STAT84 )
      { S7_Templates := "SrcType := Real"; S7_GenerateENO := "TRUE" } Sub(in1 := "DB GRUPO 1".STAT138.STAT141, in2 := 10.0, out => #RASQ_R)
      { S7_Templates := "SrcType := Real"; S7_GenerateENO := "TRUE" } Sub(in1 := "DB GRUPO 1".STAT138.STAT141, in2 := 8.0, out => #RASQ_R2)
      wire#w2
      I_Contact( "DB GRUPO 1".STAT96.STAT118 )
      { S7_Templates := "SrcType := Real" } LT_Contact(in1 := "DB GRUPO 1".STAT154.STAT157, in2 := #RASQ_R)
      S_Coil( "DB GRUPO 1".STAT96.STAT118 )
   END_RUNG
   RUNG wire#w2
      { S7_Templates := "SrcType := Real" } LT_Contact(in1 := #RASQ_R2, in2 := "DB GRUPO 1".STAT154.STAT157)
      R_Coil( "DB GRUPO 1".STAT96.STAT118 )
   END_RUNG
   RUNG wire#w1
      Contact( "DB GRUPO 1".STAT96.STAT118 )
      Coil( "Q320" )
   END_RUNG
   RUNG wire#w1
      I_Contact( "DB GRUPO 1".STAT48.STAT84 )
      R_Coil( "DB GRUPO 1".STAT96.STAT118 )
   END_RUNG
   // the same network as SCL:
   // ENO of a box is taken as its EN; it also drops when the box reports an error
   IF "DB PRINCIPAL".AUXILIARES.SEMPRE_1 THEN
       #RASQ_DI := INT_TO_DINT("P_PIW304":P);
       "DB GRUPO 1".STAT154.STAT157 := DINT_TO_REAL(#RASQ_DI);
   END_IF;
   #_w1 := "DB PRINCIPAL".AUXILIARES.SEMPRE_1 AND "DB GRUPO 1".STAT48.STAT84;
   IF #_w1 THEN
       #RASQ_R := "DB GRUPO 1".STAT138.STAT141 - 10.0;
       #RASQ_R2 := "DB GRUPO 1".STAT138.STAT141 - 8.0;
   END_IF;
   IF #_w1 AND NOT "DB GRUPO 1".STAT96.STAT118 AND ("DB GRUPO 1".STAT154.STAT157 < #RASQ_R) THEN
       "DB GRUPO 1".STAT96.STAT118 := TRUE;
   END_IF;
   IF #_w1 AND (#RASQ_R2 < "DB GRUPO 1".STAT154.STAT157) THEN "DB GRUPO 1".STAT96.STAT118 := FALSE; END_IF;
   "Q320" := "DB PRINCIPAL".AUXILIARES.SEMPRE_1 AND "DB GRUPO 1".STAT96.STAT118;
   IF "DB PRINCIPAL".AUXILIARES.SEMPRE_1 AND NOT "DB GRUPO 1".STAT48.STAT84 THEN
       "DB GRUPO 1".STAT96.STAT118 := FALSE;
   END_IF;
END_REGION

REGION Network 37: R3 - TEMPERATURA 2 LAVAGEM 1
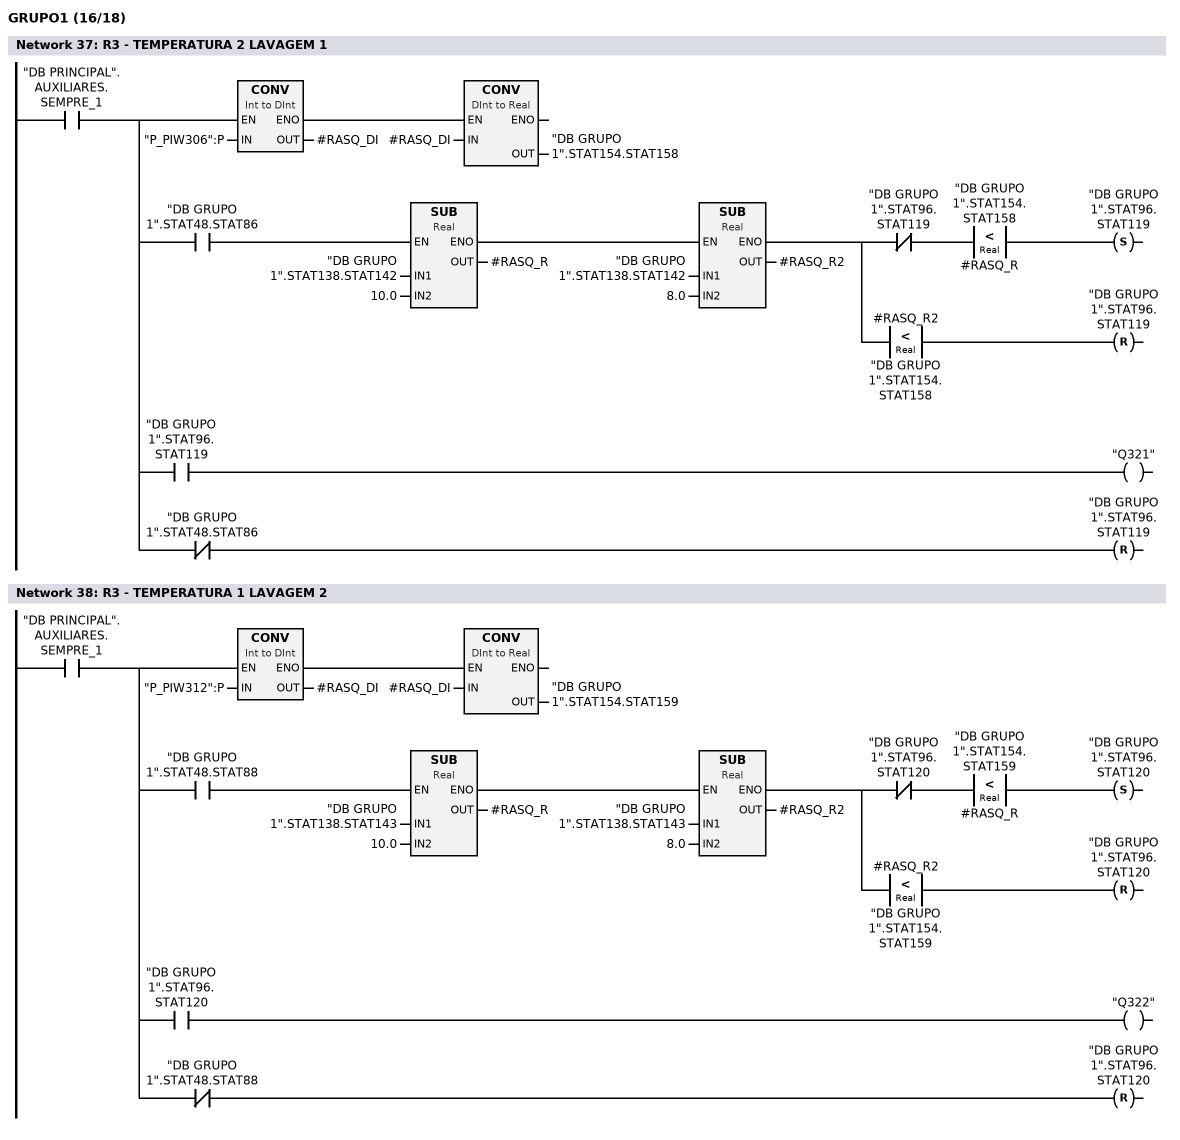
   RUNG wire#powerrail
      Contact( "DB PRINCIPAL".AUXILIARES.SEMPRE_1 )
      wire#w1
      { S7_Templates := "[SrcType := Int, DestType := DInt]"; S7_GenerateENO := "TRUE" } Convert(in := "P_PIW306":P, out => #RASQ_DI)
      { S7_Templates := "[SrcType := DInt, DestType := Real]"; S7_GenerateENO := "TRUE" } Convert(in := #RASQ_DI, out => "DB GRUPO 1".STAT154.STAT158)
   END_RUNG
   RUNG wire#w1
      Contact( "DB GRUPO 1".STAT48.STAT86 )
      { S7_Templates := "SrcType := Real"; S7_GenerateENO := "TRUE" } Sub(in1 := "DB GRUPO 1".STAT138.STAT142, in2 := 10.0, out => #RASQ_R)
      { S7_Templates := "SrcType := Real"; S7_GenerateENO := "TRUE" } Sub(in1 := "DB GRUPO 1".STAT138.STAT142, in2 := 8.0, out => #RASQ_R2)
      wire#w2
      I_Contact( "DB GRUPO 1".STAT96.STAT119 )
      { S7_Templates := "SrcType := Real" } LT_Contact(in1 := "DB GRUPO 1".STAT154.STAT158, in2 := #RASQ_R)
      S_Coil( "DB GRUPO 1".STAT96.STAT119 )
   END_RUNG
   RUNG wire#w2
      { S7_Templates := "SrcType := Real" } LT_Contact(in1 := #RASQ_R2, in2 := "DB GRUPO 1".STAT154.STAT158)
      R_Coil( "DB GRUPO 1".STAT96.STAT119 )
   END_RUNG
   RUNG wire#w1
      Contact( "DB GRUPO 1".STAT96.STAT119 )
      Coil( "Q321" )
   END_RUNG
   RUNG wire#w1
      I_Contact( "DB GRUPO 1".STAT48.STAT86 )
      R_Coil( "DB GRUPO 1".STAT96.STAT119 )
   END_RUNG
   // the same network as SCL:
   // ENO of a box is taken as its EN; it also drops when the box reports an error
   IF "DB PRINCIPAL".AUXILIARES.SEMPRE_1 THEN
       #RASQ_DI := INT_TO_DINT("P_PIW306":P);
       "DB GRUPO 1".STAT154.STAT158 := DINT_TO_REAL(#RASQ_DI);
   END_IF;
   #_w1 := "DB PRINCIPAL".AUXILIARES.SEMPRE_1 AND "DB GRUPO 1".STAT48.STAT86;
   IF #_w1 THEN
       #RASQ_R := "DB GRUPO 1".STAT138.STAT142 - 10.0;
       #RASQ_R2 := "DB GRUPO 1".STAT138.STAT142 - 8.0;
   END_IF;
   IF #_w1 AND NOT "DB GRUPO 1".STAT96.STAT119 AND ("DB GRUPO 1".STAT154.STAT158 < #RASQ_R) THEN
       "DB GRUPO 1".STAT96.STAT119 := TRUE;
   END_IF;
   IF #_w1 AND (#RASQ_R2 < "DB GRUPO 1".STAT154.STAT158) THEN "DB GRUPO 1".STAT96.STAT119 := FALSE; END_IF;
   "Q321" := "DB PRINCIPAL".AUXILIARES.SEMPRE_1 AND "DB GRUPO 1".STAT96.STAT119;
   IF "DB PRINCIPAL".AUXILIARES.SEMPRE_1 AND NOT "DB GRUPO 1".STAT48.STAT86 THEN
       "DB GRUPO 1".STAT96.STAT119 := FALSE;
   END_IF;
END_REGION

REGION Network 38: R3 - TEMPERATURA 1 LAVAGEM 2
   RUNG wire#powerrail
      Contact( "DB PRINCIPAL".AUXILIARES.SEMPRE_1 )
      wire#w1
      { S7_Templates := "[SrcType := Int, DestType := DInt]"; S7_GenerateENO := "TRUE" } Convert(in := "P_PIW312":P, out => #RASQ_DI)
      { S7_Templates := "[SrcType := DInt, DestType := Real]"; S7_GenerateENO := "TRUE" } Convert(in := #RASQ_DI, out => "DB GRUPO 1".STAT154.STAT159)
   END_RUNG
   RUNG wire#w1
      Contact( "DB GRUPO 1".STAT48.STAT88 )
      { S7_Templates := "SrcType := Real"; S7_GenerateENO := "TRUE" } Sub(in1 := "DB GRUPO 1".STAT138.STAT143, in2 := 10.0, out => #RASQ_R)
      { S7_Templates := "SrcType := Real"; S7_GenerateENO := "TRUE" } Sub(in1 := "DB GRUPO 1".STAT138.STAT143, in2 := 8.0, out => #RASQ_R2)
      wire#w2
      I_Contact( "DB GRUPO 1".STAT96.STAT120 )
      { S7_Templates := "SrcType := Real" } LT_Contact(in1 := "DB GRUPO 1".STAT154.STAT159, in2 := #RASQ_R)
      S_Coil( "DB GRUPO 1".STAT96.STAT120 )
   END_RUNG
   RUNG wire#w2
      { S7_Templates := "SrcType := Real" } LT_Contact(in1 := #RASQ_R2, in2 := "DB GRUPO 1".STAT154.STAT159)
      R_Coil( "DB GRUPO 1".STAT96.STAT120 )
   END_RUNG
   RUNG wire#w1
      Contact( "DB GRUPO 1".STAT96.STAT120 )
      Coil( "Q322" )
   END_RUNG
   RUNG wire#w1
      I_Contact( "DB GRUPO 1".STAT48.STAT88 )
      R_Coil( "DB GRUPO 1".STAT96.STAT120 )
   END_RUNG
   // the same network as SCL:
   // ENO of a box is taken as its EN; it also drops when the box reports an error
   IF "DB PRINCIPAL".AUXILIARES.SEMPRE_1 THEN
       #RASQ_DI := INT_TO_DINT("P_PIW312":P);
       "DB GRUPO 1".STAT154.STAT159 := DINT_TO_REAL(#RASQ_DI);
   END_IF;
   #_w1 := "DB PRINCIPAL".AUXILIARES.SEMPRE_1 AND "DB GRUPO 1".STAT48.STAT88;
   IF #_w1 THEN
       #RASQ_R := "DB GRUPO 1".STAT138.STAT143 - 10.0;
       #RASQ_R2 := "DB GRUPO 1".STAT138.STAT143 - 8.0;
   END_IF;
   IF #_w1 AND NOT "DB GRUPO 1".STAT96.STAT120 AND ("DB GRUPO 1".STAT154.STAT159 < #RASQ_R) THEN
       "DB GRUPO 1".STAT96.STAT120 := TRUE;
   END_IF;
   IF #_w1 AND (#RASQ_R2 < "DB GRUPO 1".STAT154.STAT159) THEN "DB GRUPO 1".STAT96.STAT120 := FALSE; END_IF;
   "Q322" := "DB PRINCIPAL".AUXILIARES.SEMPRE_1 AND "DB GRUPO 1".STAT96.STAT120;
   IF "DB PRINCIPAL".AUXILIARES.SEMPRE_1 AND NOT "DB GRUPO 1".STAT48.STAT88 THEN
       "DB GRUPO 1".STAT96.STAT120 := FALSE;
   END_IF;
END_REGION

REGION Network 39: R3 - TEMPERATURA 2 LAVAGEM 2
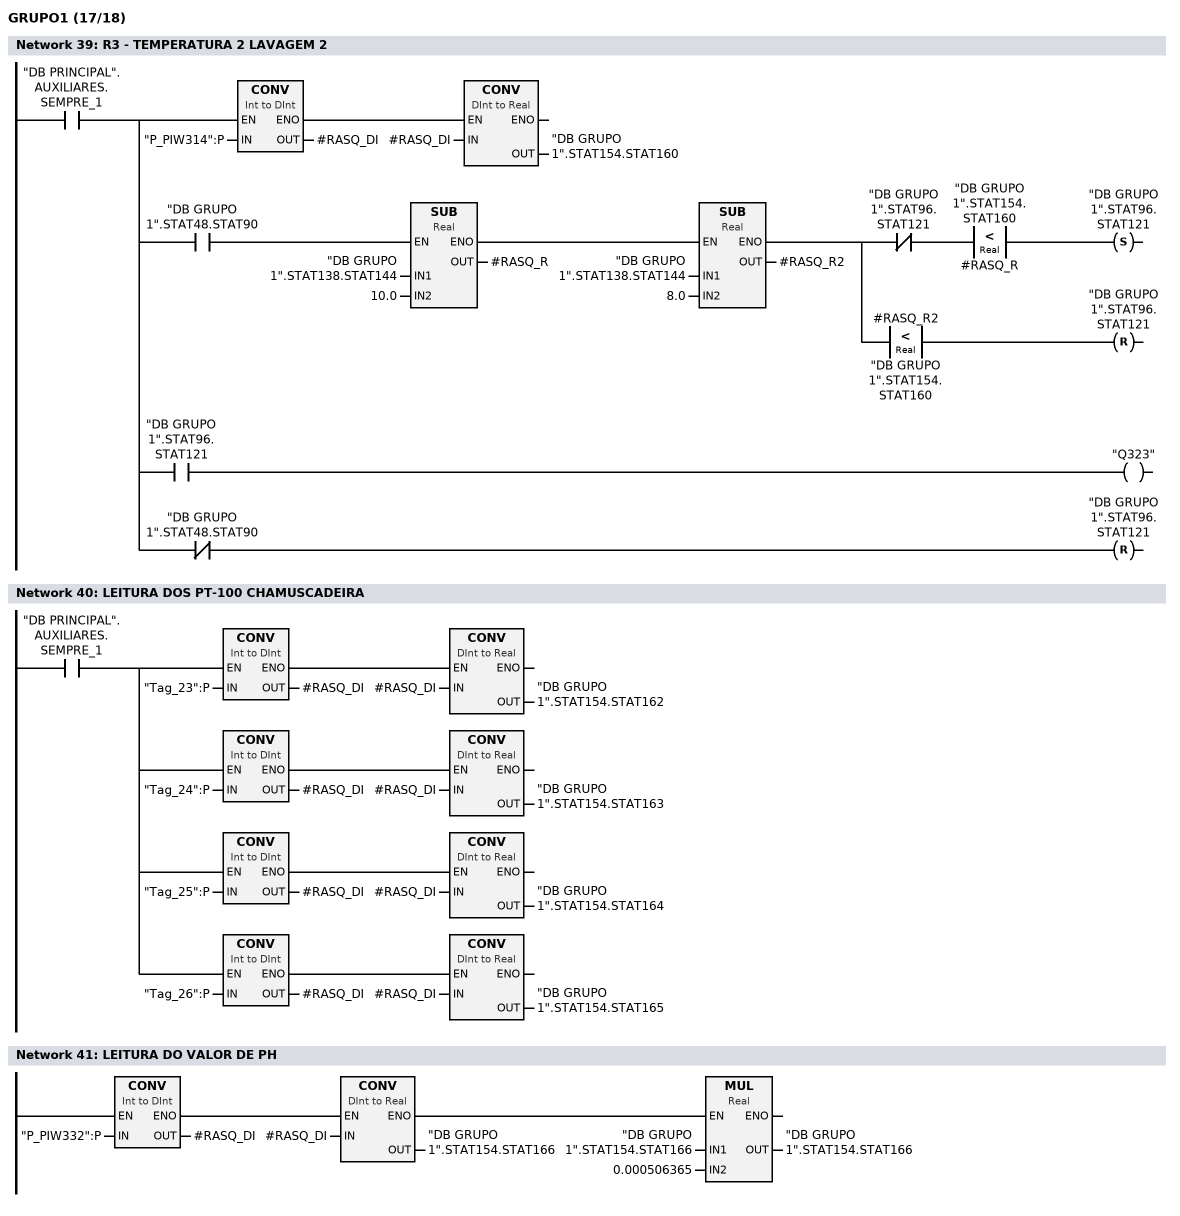
   RUNG wire#powerrail
      Contact( "DB PRINCIPAL".AUXILIARES.SEMPRE_1 )
      wire#w1
      { S7_Templates := "[SrcType := Int, DestType := DInt]"; S7_GenerateENO := "TRUE" } Convert(in := "P_PIW314":P, out => #RASQ_DI)
      { S7_Templates := "[SrcType := DInt, DestType := Real]"; S7_GenerateENO := "TRUE" } Convert(in := #RASQ_DI, out => "DB GRUPO 1".STAT154.STAT160)
   END_RUNG
   RUNG wire#w1
      Contact( "DB GRUPO 1".STAT48.STAT90 )
      { S7_Templates := "SrcType := Real"; S7_GenerateENO := "TRUE" } Sub(in1 := "DB GRUPO 1".STAT138.STAT144, in2 := 10.0, out => #RASQ_R)
      { S7_Templates := "SrcType := Real"; S7_GenerateENO := "TRUE" } Sub(in1 := "DB GRUPO 1".STAT138.STAT144, in2 := 8.0, out => #RASQ_R2)
      wire#w2
      I_Contact( "DB GRUPO 1".STAT96.STAT121 )
      { S7_Templates := "SrcType := Real" } LT_Contact(in1 := "DB GRUPO 1".STAT154.STAT160, in2 := #RASQ_R)
      S_Coil( "DB GRUPO 1".STAT96.STAT121 )
   END_RUNG
   RUNG wire#w2
      { S7_Templates := "SrcType := Real" } LT_Contact(in1 := #RASQ_R2, in2 := "DB GRUPO 1".STAT154.STAT160)
      R_Coil( "DB GRUPO 1".STAT96.STAT121 )
   END_RUNG
   RUNG wire#w1
      Contact( "DB GRUPO 1".STAT96.STAT121 )
      Coil( "Q323" )
   END_RUNG
   RUNG wire#w1
      I_Contact( "DB GRUPO 1".STAT48.STAT90 )
      R_Coil( "DB GRUPO 1".STAT96.STAT121 )
   END_RUNG
   // the same network as SCL:
   // ENO of a box is taken as its EN; it also drops when the box reports an error
   IF "DB PRINCIPAL".AUXILIARES.SEMPRE_1 THEN
       #RASQ_DI := INT_TO_DINT("P_PIW314":P);
       "DB GRUPO 1".STAT154.STAT160 := DINT_TO_REAL(#RASQ_DI);
   END_IF;
   #_w1 := "DB PRINCIPAL".AUXILIARES.SEMPRE_1 AND "DB GRUPO 1".STAT48.STAT90;
   IF #_w1 THEN
       #RASQ_R := "DB GRUPO 1".STAT138.STAT144 - 10.0;
       #RASQ_R2 := "DB GRUPO 1".STAT138.STAT144 - 8.0;
   END_IF;
   IF #_w1 AND NOT "DB GRUPO 1".STAT96.STAT121 AND ("DB GRUPO 1".STAT154.STAT160 < #RASQ_R) THEN
       "DB GRUPO 1".STAT96.STAT121 := TRUE;
   END_IF;
   IF #_w1 AND (#RASQ_R2 < "DB GRUPO 1".STAT154.STAT160) THEN "DB GRUPO 1".STAT96.STAT121 := FALSE; END_IF;
   "Q323" := "DB PRINCIPAL".AUXILIARES.SEMPRE_1 AND "DB GRUPO 1".STAT96.STAT121;
   IF "DB PRINCIPAL".AUXILIARES.SEMPRE_1 AND NOT "DB GRUPO 1".STAT48.STAT90 THEN
       "DB GRUPO 1".STAT96.STAT121 := FALSE;
   END_IF;
END_REGION

REGION Network 40: LEITURA DOS PT-100 CHAMUSCADEIRA
   RUNG wire#powerrail
      Contact( "DB PRINCIPAL".AUXILIARES.SEMPRE_1 )
      wire#w1
      { S7_Templates := "[SrcType := Int, DestType := DInt]"; S7_GenerateENO := "TRUE" } Convert(in := "Tag_23":P, out => #RASQ_DI)
      { S7_Templates := "[SrcType := DInt, DestType := Real]"; S7_GenerateENO := "TRUE" } Convert(in := #RASQ_DI, out => "DB GRUPO 1".STAT154.STAT162)
   END_RUNG
   RUNG wire#w1
      { S7_Templates := "[SrcType := Int, DestType := DInt]"; S7_GenerateENO := "TRUE" } Convert(in := "Tag_24":P, out => #RASQ_DI)
      { S7_Templates := "[SrcType := DInt, DestType := Real]"; S7_GenerateENO := "TRUE" } Convert(in := #RASQ_DI, out => "DB GRUPO 1".STAT154.STAT163)
   END_RUNG
   RUNG wire#w1
      { S7_Templates := "[SrcType := Int, DestType := DInt]"; S7_GenerateENO := "TRUE" } Convert(in := "Tag_25":P, out => #RASQ_DI)
      { S7_Templates := "[SrcType := DInt, DestType := Real]"; S7_GenerateENO := "TRUE" } Convert(in := #RASQ_DI, out => "DB GRUPO 1".STAT154.STAT164)
   END_RUNG
   RUNG wire#w1
      { S7_Templates := "[SrcType := Int, DestType := DInt]"; S7_GenerateENO := "TRUE" } Convert(in := "Tag_26":P, out => #RASQ_DI)
      { S7_Templates := "[SrcType := DInt, DestType := Real]"; S7_GenerateENO := "TRUE" } Convert(in := #RASQ_DI, out => "DB GRUPO 1".STAT154.STAT165)
   END_RUNG
   // the same network as SCL:
   // ENO of a box is taken as its EN; it also drops when the box reports an error
   IF "DB PRINCIPAL".AUXILIARES.SEMPRE_1 THEN
       #RASQ_DI := INT_TO_DINT("Tag_23":P);
       "DB GRUPO 1".STAT154.STAT162 := DINT_TO_REAL(#RASQ_DI);
       #RASQ_DI := INT_TO_DINT("Tag_24":P);
       "DB GRUPO 1".STAT154.STAT163 := DINT_TO_REAL(#RASQ_DI);
       #RASQ_DI := INT_TO_DINT("Tag_25":P);
       "DB GRUPO 1".STAT154.STAT164 := DINT_TO_REAL(#RASQ_DI);
       #RASQ_DI := INT_TO_DINT("Tag_26":P);
       "DB GRUPO 1".STAT154.STAT165 := DINT_TO_REAL(#RASQ_DI);
   END_IF;
END_REGION

REGION Network 41: LEITURA DO VALOR DE PH
   RUNG wire#powerrail
      { S7_Templates := "[SrcType := Int, DestType := DInt]"; S7_GenerateENO := "TRUE" } Convert(in := "P_PIW332":P, out => #RASQ_DI)
      { S7_Templates := "[SrcType := DInt, DestType := Real]"; S7_GenerateENO := "TRUE" } Convert(in := #RASQ_DI, out => "DB GRUPO 1".STAT154.STAT166)
      { S7_Templates := "SrcType := Real"; S7_GenerateENO := "TRUE" } Mul(in1 := "DB GRUPO 1".STAT154.STAT166, in2 := 0.000506365, out => "DB GRUPO 1".STAT154.STAT166)
   END_RUNG
   // the same network as SCL:
   // ENO of a box is taken as its EN; it also drops when the box reports an error
   #RASQ_DI := INT_TO_DINT("P_PIW332":P);
   "DB GRUPO 1".STAT154.STAT166 := DINT_TO_REAL(#RASQ_DI);
   "DB GRUPO 1".STAT154.STAT166 := "DB GRUPO 1".STAT154.STAT166 * 0.000506365;
END_REGION

REGION Network 42: ACIONA ALARMES
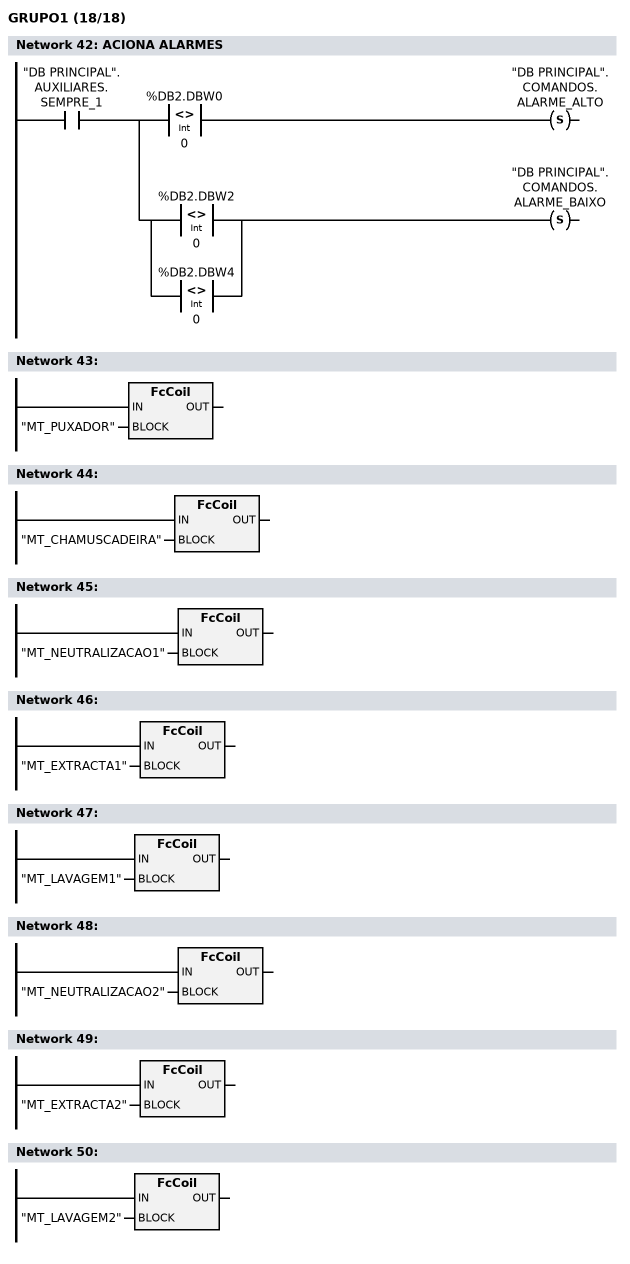
   RUNG wire#powerrail
      Contact( "DB PRINCIPAL".AUXILIARES.SEMPRE_1 )
      wire#w1
      { S7_Templates := "SrcType := Int" } NE_Contact(in1 := %DB2.DBW0, in2 := 0)
      S_Coil( "DB PRINCIPAL".COMANDOS.ALARME_ALTO )
   END_RUNG
   RUNG wire#w1
      { S7_Templates := "SrcType := Int" } NE_Contact(in1 := %DB2.DBW2, in2 := 0)
      wire#w2
      S_Coil( "DB PRINCIPAL".COMANDOS.ALARME_BAIXO )
   END_RUNG
   RUNG wire#w1
      { S7_Templates := "SrcType := Int" } NE_Contact(in1 := %DB2.DBW4, in2 := 0)
   END_RUNG wire#w2
   // the same network as SCL:
   IF "DB PRINCIPAL".AUXILIARES.SEMPRE_1 AND (%DB2.DBW0 <> 0) THEN
       "DB PRINCIPAL".COMANDOS.ALARME_ALTO := TRUE;
   END_IF;
   IF "DB PRINCIPAL".AUXILIARES.SEMPRE_1 AND ((%DB2.DBW2 <> 0) OR (%DB2.DBW4 <> 0)) THEN
       "DB PRINCIPAL".COMANDOS.ALARME_BAIXO := TRUE;
   END_IF;
END_REGION

REGION Network 43
   // no SCL statement known for FcCoil: written as a call
   FcCoil(block := "MT_PUXADOR", in := TRUE);
END_REGION

REGION Network 44
   // no SCL statement known for FcCoil: written as a call
   FcCoil(block := "MT_CHAMUSCADEIRA", in := TRUE);
END_REGION

REGION Network 45
   // no SCL statement known for FcCoil: written as a call
   FcCoil(block := "MT_NEUTRALIZACAO1", in := TRUE);
END_REGION

REGION Network 46
   // no SCL statement known for FcCoil: written as a call
   FcCoil(block := "MT_EXTRACTA1", in := TRUE);
END_REGION

REGION Network 47
   // no SCL statement known for FcCoil: written as a call
   FcCoil(block := "MT_LAVAGEM1", in := TRUE);
END_REGION

REGION Network 48
   // no SCL statement known for FcCoil: written as a call
   FcCoil(block := "MT_NEUTRALIZACAO2", in := TRUE);
END_REGION

REGION Network 49
   // no SCL statement known for FcCoil: written as a call
   FcCoil(block := "MT_EXTRACTA2", in := TRUE);
END_REGION

REGION Network 50
   // no SCL statement known for FcCoil: written as a call
   FcCoil(block := "MT_LAVAGEM2", in := TRUE);
END_REGION
END_FUNCTION

FUNCTION "GRUPO2" : Void   // FC3, LAD
{ S7_Optimized_Access := 'FALSE' }
VERSION : 0.1
   VAR_TEMP
      RASQ_DI : DInt;
      RASQ_R : Real;
   END_VAR
   VAR_TEMP   // added for the SCL form of the ladder/FBD networks
      _w1 : Bool;
   END_VAR
BEGIN

REGION Network 1: RESET DO ALARMES
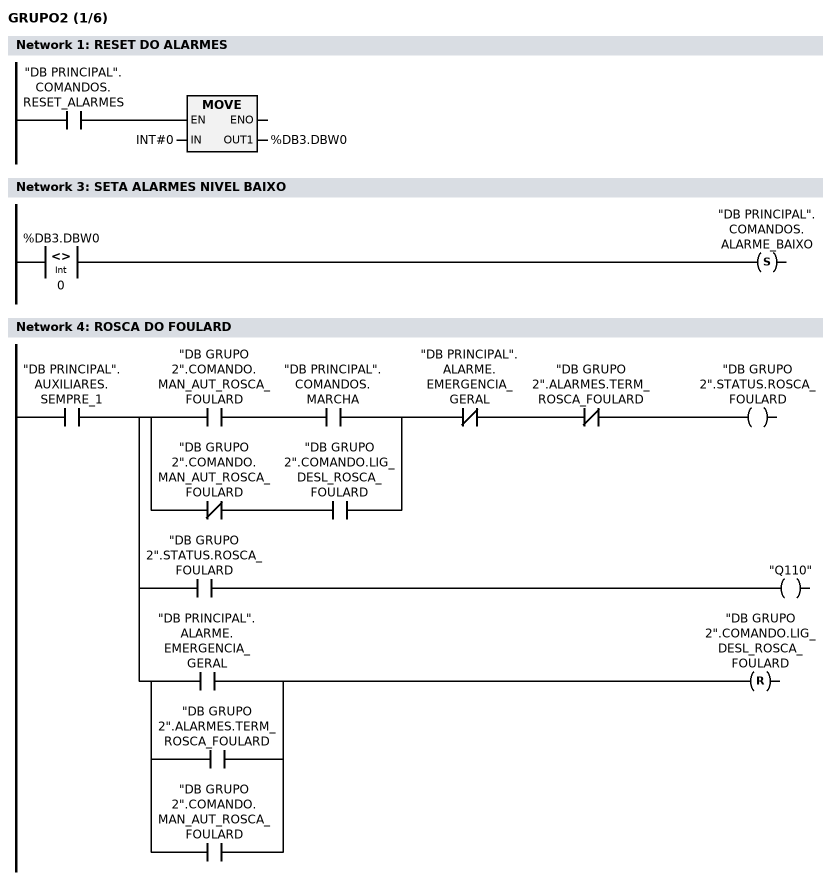
   RUNG wire#powerrail
      Contact( "DB PRINCIPAL".COMANDOS.RESET_ALARMES )
      { S7_GenerateENO := "TRUE" } Move(in := INT#0, out1 => %DB3.DBW0)
   END_RUNG
   // the same network as SCL:
   IF "DB PRINCIPAL".COMANDOS.RESET_ALARMES THEN %DB3.DBW0 := INT#0; END_IF;
END_REGION

REGION Network 2 (STL): ALARMES
         A     "DB PRINCIPAL".AUXILIARES.SEMPRE_1;
         =     <??.?>;
         A     <??.?>;
         A     "I111";
         =     "DB GRUPO 2".ALARMES.TERM_ROSCA_FOULARD;
         A     <??.?>;
         A     "I116";
         =     "DB GRUPO 2".ALARMES.TERM_EXAUSTOR_SECA1;
         A     <??.?>;
         A     "I117";
         =     "DB GRUPO 2".ALARMES.TERM_EXAUSTOR_SECA2;
         A     <??.?>;
         A     "I120";
         =     "DB GRUPO 2".ALARMES.TERM_EXAUSTOR_SECA3;
         A     <??.?>;
         A     "I121";
         =     "DB GRUPO 2".ALARMES.TERM_EXAUSTOR_SECA4;
         NOP   0;
END_REGION

REGION Network 3: SETA ALARMES NIVEL BAIXO
   RUNG wire#powerrail
      { S7_Templates := "SrcType := Int" } NE_Contact(in1 := %DB3.DBW0, in2 := 0)
      S_Coil( "DB PRINCIPAL".COMANDOS.ALARME_BAIXO )
   END_RUNG
   // the same network as SCL:
   IF %DB3.DBW0 <> 0 THEN "DB PRINCIPAL".COMANDOS.ALARME_BAIXO := TRUE; END_IF;
END_REGION

REGION Network 4: ROSCA DO FOULARD
   RUNG wire#powerrail
      Contact( "DB PRINCIPAL".AUXILIARES.SEMPRE_1 )
      wire#w1
      Contact( "DB GRUPO 2".COMANDO.MAN_AUT_ROSCA_FOULARD )
      Contact( "DB PRINCIPAL".COMANDOS.MARCHA )
      wire#w2
      I_Contact( "DB PRINCIPAL".ALARME.EMERGENCIA_GERAL )
      I_Contact( "DB GRUPO 2".ALARMES.TERM_ROSCA_FOULARD )
      Coil( "DB GRUPO 2".STATUS.ROSCA_FOULARD )
   END_RUNG
   RUNG wire#w1
      I_Contact( "DB GRUPO 2".COMANDO.MAN_AUT_ROSCA_FOULARD )
      Contact( "DB GRUPO 2".COMANDO.LIG_DESL_ROSCA_FOULARD )
   END_RUNG wire#w2
   RUNG wire#w1
      Contact( "DB GRUPO 2".STATUS.ROSCA_FOULARD )
      Coil( "Q110" )
   END_RUNG
   RUNG wire#w1
      Contact( "DB PRINCIPAL".ALARME.EMERGENCIA_GERAL )
      wire#w3
      R_Coil( "DB GRUPO 2".COMANDO.LIG_DESL_ROSCA_FOULARD )
   END_RUNG
   RUNG wire#w1
      Contact( "DB GRUPO 2".ALARMES.TERM_ROSCA_FOULARD )
   END_RUNG wire#w3
   RUNG wire#w1
      Contact( "DB GRUPO 2".COMANDO.MAN_AUT_ROSCA_FOULARD )
   END_RUNG wire#w3
   // the same network as SCL:
   "DB GRUPO 2".STATUS.ROSCA_FOULARD := "DB PRINCIPAL".AUXILIARES.SEMPRE_1 AND (("DB GRUPO 2".COMANDO.MAN_AUT_ROSCA_FOULARD AND "DB PRINCIPAL".COMANDOS.MARCHA) OR (NOT "DB GRUPO 2".COMANDO.MAN_AUT_ROSCA_FOULARD AND "DB GRUPO 2".COMANDO.LIG_DESL_ROSCA_FOULARD)) AND NOT "DB PRINCIPAL".ALARME.EMERGENCIA_GERAL AND NOT "DB GRUPO 2".ALARMES.TERM_ROSCA_FOULARD;
   "Q110" := "DB PRINCIPAL".AUXILIARES.SEMPRE_1 AND "DB GRUPO 2".STATUS.ROSCA_FOULARD;
   IF "DB PRINCIPAL".AUXILIARES.SEMPRE_1 AND ("DB PRINCIPAL".ALARME.EMERGENCIA_GERAL OR "DB GRUPO 2".ALARMES.TERM_ROSCA_FOULARD OR "DB GRUPO 2".COMANDO.MAN_AUT_ROSCA_FOULARD) THEN
       "DB GRUPO 2".COMANDO.LIG_DESL_ROSCA_FOULARD := FALSE;
   END_IF;
END_REGION

REGION Network 5: NIVEL DO FOULARD
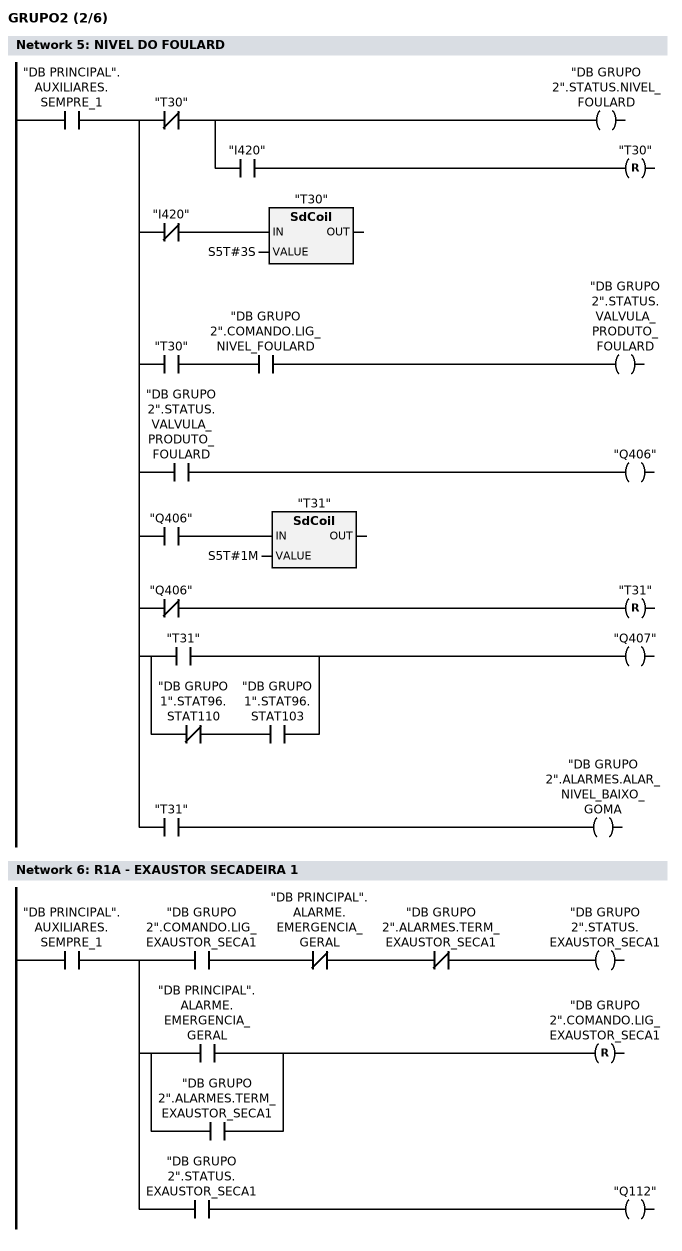
   // no SCL statement known for SdCoil: written as a call
   "DB GRUPO 2".STATUS.NIVEL_FOULARD := "DB PRINCIPAL".AUXILIARES.SEMPRE_1 AND NOT "T30";
   IF "DB GRUPO 2".STATUS.NIVEL_FOULARD AND "I420" THEN "T30" := FALSE; END_IF;
   #_w1 := "DB PRINCIPAL".AUXILIARES.SEMPRE_1;
   SdCoil(value := S5T#3S, operand := "T30", in := "DB PRINCIPAL".AUXILIARES.SEMPRE_1 AND NOT "I420");
   "DB GRUPO 2".STATUS.VALVULA_PRODUTO_FOULARD := #_w1 AND "T30" AND "DB GRUPO 2".COMANDO.LIG_NIVEL_FOULARD;
   "Q406" := #_w1 AND "DB GRUPO 2".STATUS.VALVULA_PRODUTO_FOULARD;
   SdCoil(value := S5T#1M, operand := "T31", in := #_w1 AND "Q406");
   IF #_w1 AND NOT "Q406" THEN "T31" := FALSE; END_IF;
   "Q407" := #_w1 AND ("T31" OR (NOT "DB GRUPO 1".STAT96.STAT110 AND "DB GRUPO 1".STAT96.STAT103));
   "DB GRUPO 2".ALARMES.ALAR_NIVEL_BAIXO_GOMA := #_w1 AND "T31";
END_REGION

REGION Network 6: R1A - EXAUSTOR SECADEIRA 1
   RUNG wire#powerrail
      Contact( "DB PRINCIPAL".AUXILIARES.SEMPRE_1 )
      wire#w1
      Contact( "DB GRUPO 2".COMANDO.LIG_EXAUSTOR_SECA1 )
      I_Contact( "DB PRINCIPAL".ALARME.EMERGENCIA_GERAL )
      I_Contact( "DB GRUPO 2".ALARMES.TERM_EXAUSTOR_SECA1 )
      Coil( "DB GRUPO 2".STATUS.EXAUSTOR_SECA1 )
   END_RUNG
   RUNG wire#w1
      Contact( "DB PRINCIPAL".ALARME.EMERGENCIA_GERAL )
      wire#w2
      R_Coil( "DB GRUPO 2".COMANDO.LIG_EXAUSTOR_SECA1 )
   END_RUNG
   RUNG wire#w1
      Contact( "DB GRUPO 2".ALARMES.TERM_EXAUSTOR_SECA1 )
   END_RUNG wire#w2
   RUNG wire#w1
      Contact( "DB GRUPO 2".STATUS.EXAUSTOR_SECA1 )
      Coil( "Q112" )
   END_RUNG
   // the same network as SCL:
   "DB GRUPO 2".STATUS.EXAUSTOR_SECA1 := "DB PRINCIPAL".AUXILIARES.SEMPRE_1 AND "DB GRUPO 2".COMANDO.LIG_EXAUSTOR_SECA1 AND NOT "DB PRINCIPAL".ALARME.EMERGENCIA_GERAL AND NOT "DB GRUPO 2".ALARMES.TERM_EXAUSTOR_SECA1;
   IF "DB PRINCIPAL".AUXILIARES.SEMPRE_1 AND ("DB PRINCIPAL".ALARME.EMERGENCIA_GERAL OR "DB GRUPO 2".ALARMES.TERM_EXAUSTOR_SECA1) THEN
       "DB GRUPO 2".COMANDO.LIG_EXAUSTOR_SECA1 := FALSE;
   END_IF;
   "Q112" := "DB PRINCIPAL".AUXILIARES.SEMPRE_1 AND "DB GRUPO 2".STATUS.EXAUSTOR_SECA1;
END_REGION

REGION Network 7: R1A - EXAUSTOR SECADEIRA 2
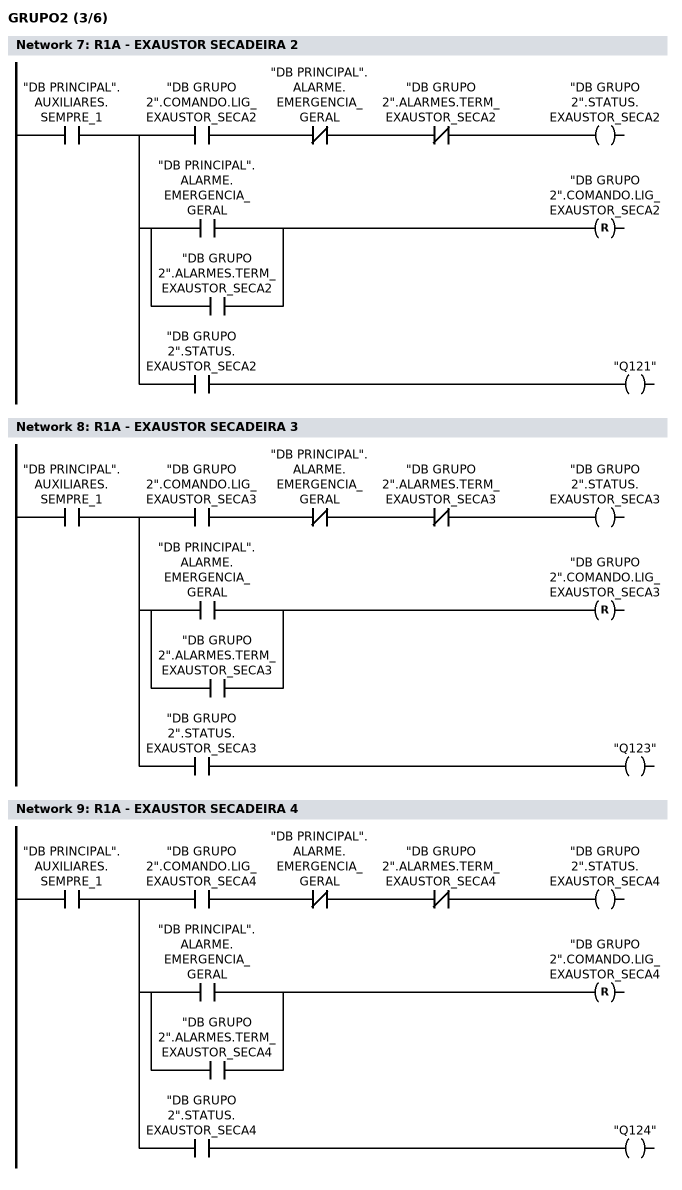
   RUNG wire#powerrail
      Contact( "DB PRINCIPAL".AUXILIARES.SEMPRE_1 )
      wire#w1
      Contact( "DB GRUPO 2".COMANDO.LIG_EXAUSTOR_SECA2 )
      I_Contact( "DB PRINCIPAL".ALARME.EMERGENCIA_GERAL )
      I_Contact( "DB GRUPO 2".ALARMES.TERM_EXAUSTOR_SECA2 )
      Coil( "DB GRUPO 2".STATUS.EXAUSTOR_SECA2 )
   END_RUNG
   RUNG wire#w1
      Contact( "DB PRINCIPAL".ALARME.EMERGENCIA_GERAL )
      wire#w2
      R_Coil( "DB GRUPO 2".COMANDO.LIG_EXAUSTOR_SECA2 )
   END_RUNG
   RUNG wire#w1
      Contact( "DB GRUPO 2".ALARMES.TERM_EXAUSTOR_SECA2 )
   END_RUNG wire#w2
   RUNG wire#w1
      Contact( "DB GRUPO 2".STATUS.EXAUSTOR_SECA2 )
      Coil( "Q121" )
   END_RUNG
   // the same network as SCL:
   "DB GRUPO 2".STATUS.EXAUSTOR_SECA2 := "DB PRINCIPAL".AUXILIARES.SEMPRE_1 AND "DB GRUPO 2".COMANDO.LIG_EXAUSTOR_SECA2 AND NOT "DB PRINCIPAL".ALARME.EMERGENCIA_GERAL AND NOT "DB GRUPO 2".ALARMES.TERM_EXAUSTOR_SECA2;
   IF "DB PRINCIPAL".AUXILIARES.SEMPRE_1 AND ("DB PRINCIPAL".ALARME.EMERGENCIA_GERAL OR "DB GRUPO 2".ALARMES.TERM_EXAUSTOR_SECA2) THEN
       "DB GRUPO 2".COMANDO.LIG_EXAUSTOR_SECA2 := FALSE;
   END_IF;
   "Q121" := "DB PRINCIPAL".AUXILIARES.SEMPRE_1 AND "DB GRUPO 2".STATUS.EXAUSTOR_SECA2;
END_REGION

REGION Network 8: R1A - EXAUSTOR SECADEIRA 3
   RUNG wire#powerrail
      Contact( "DB PRINCIPAL".AUXILIARES.SEMPRE_1 )
      wire#w1
      Contact( "DB GRUPO 2".COMANDO.LIG_EXAUSTOR_SECA3 )
      I_Contact( "DB PRINCIPAL".ALARME.EMERGENCIA_GERAL )
      I_Contact( "DB GRUPO 2".ALARMES.TERM_EXAUSTOR_SECA3 )
      Coil( "DB GRUPO 2".STATUS.EXAUSTOR_SECA3 )
   END_RUNG
   RUNG wire#w1
      Contact( "DB PRINCIPAL".ALARME.EMERGENCIA_GERAL )
      wire#w2
      R_Coil( "DB GRUPO 2".COMANDO.LIG_EXAUSTOR_SECA3 )
   END_RUNG
   RUNG wire#w1
      Contact( "DB GRUPO 2".ALARMES.TERM_EXAUSTOR_SECA3 )
   END_RUNG wire#w2
   RUNG wire#w1
      Contact( "DB GRUPO 2".STATUS.EXAUSTOR_SECA3 )
      Coil( "Q123" )
   END_RUNG
   // the same network as SCL:
   "DB GRUPO 2".STATUS.EXAUSTOR_SECA3 := "DB PRINCIPAL".AUXILIARES.SEMPRE_1 AND "DB GRUPO 2".COMANDO.LIG_EXAUSTOR_SECA3 AND NOT "DB PRINCIPAL".ALARME.EMERGENCIA_GERAL AND NOT "DB GRUPO 2".ALARMES.TERM_EXAUSTOR_SECA3;
   IF "DB PRINCIPAL".AUXILIARES.SEMPRE_1 AND ("DB PRINCIPAL".ALARME.EMERGENCIA_GERAL OR "DB GRUPO 2".ALARMES.TERM_EXAUSTOR_SECA3) THEN
       "DB GRUPO 2".COMANDO.LIG_EXAUSTOR_SECA3 := FALSE;
   END_IF;
   "Q123" := "DB PRINCIPAL".AUXILIARES.SEMPRE_1 AND "DB GRUPO 2".STATUS.EXAUSTOR_SECA3;
END_REGION

REGION Network 9: R1A - EXAUSTOR SECADEIRA 4
   RUNG wire#powerrail
      Contact( "DB PRINCIPAL".AUXILIARES.SEMPRE_1 )
      wire#w1
      Contact( "DB GRUPO 2".COMANDO.LIG_EXAUSTOR_SECA4 )
      I_Contact( "DB PRINCIPAL".ALARME.EMERGENCIA_GERAL )
      I_Contact( "DB GRUPO 2".ALARMES.TERM_EXAUSTOR_SECA4 )
      Coil( "DB GRUPO 2".STATUS.EXAUSTOR_SECA4 )
   END_RUNG
   RUNG wire#w1
      Contact( "DB PRINCIPAL".ALARME.EMERGENCIA_GERAL )
      wire#w2
      R_Coil( "DB GRUPO 2".COMANDO.LIG_EXAUSTOR_SECA4 )
   END_RUNG
   RUNG wire#w1
      Contact( "DB GRUPO 2".ALARMES.TERM_EXAUSTOR_SECA4 )
   END_RUNG wire#w2
   RUNG wire#w1
      Contact( "DB GRUPO 2".STATUS.EXAUSTOR_SECA4 )
      Coil( "Q124" )
   END_RUNG
   // the same network as SCL:
   "DB GRUPO 2".STATUS.EXAUSTOR_SECA4 := "DB PRINCIPAL".AUXILIARES.SEMPRE_1 AND "DB GRUPO 2".COMANDO.LIG_EXAUSTOR_SECA4 AND NOT "DB PRINCIPAL".ALARME.EMERGENCIA_GERAL AND NOT "DB GRUPO 2".ALARMES.TERM_EXAUSTOR_SECA4;
   IF "DB PRINCIPAL".AUXILIARES.SEMPRE_1 AND ("DB PRINCIPAL".ALARME.EMERGENCIA_GERAL OR "DB GRUPO 2".ALARMES.TERM_EXAUSTOR_SECA4) THEN
       "DB GRUPO 2".COMANDO.LIG_EXAUSTOR_SECA4 := FALSE;
   END_IF;
   "Q124" := "DB PRINCIPAL".AUXILIARES.SEMPRE_1 AND "DB GRUPO 2".STATUS.EXAUSTOR_SECA4;
END_REGION

REGION Network 10: R3 - TEMPERATURA TANQUE 1 DE PRODUTO
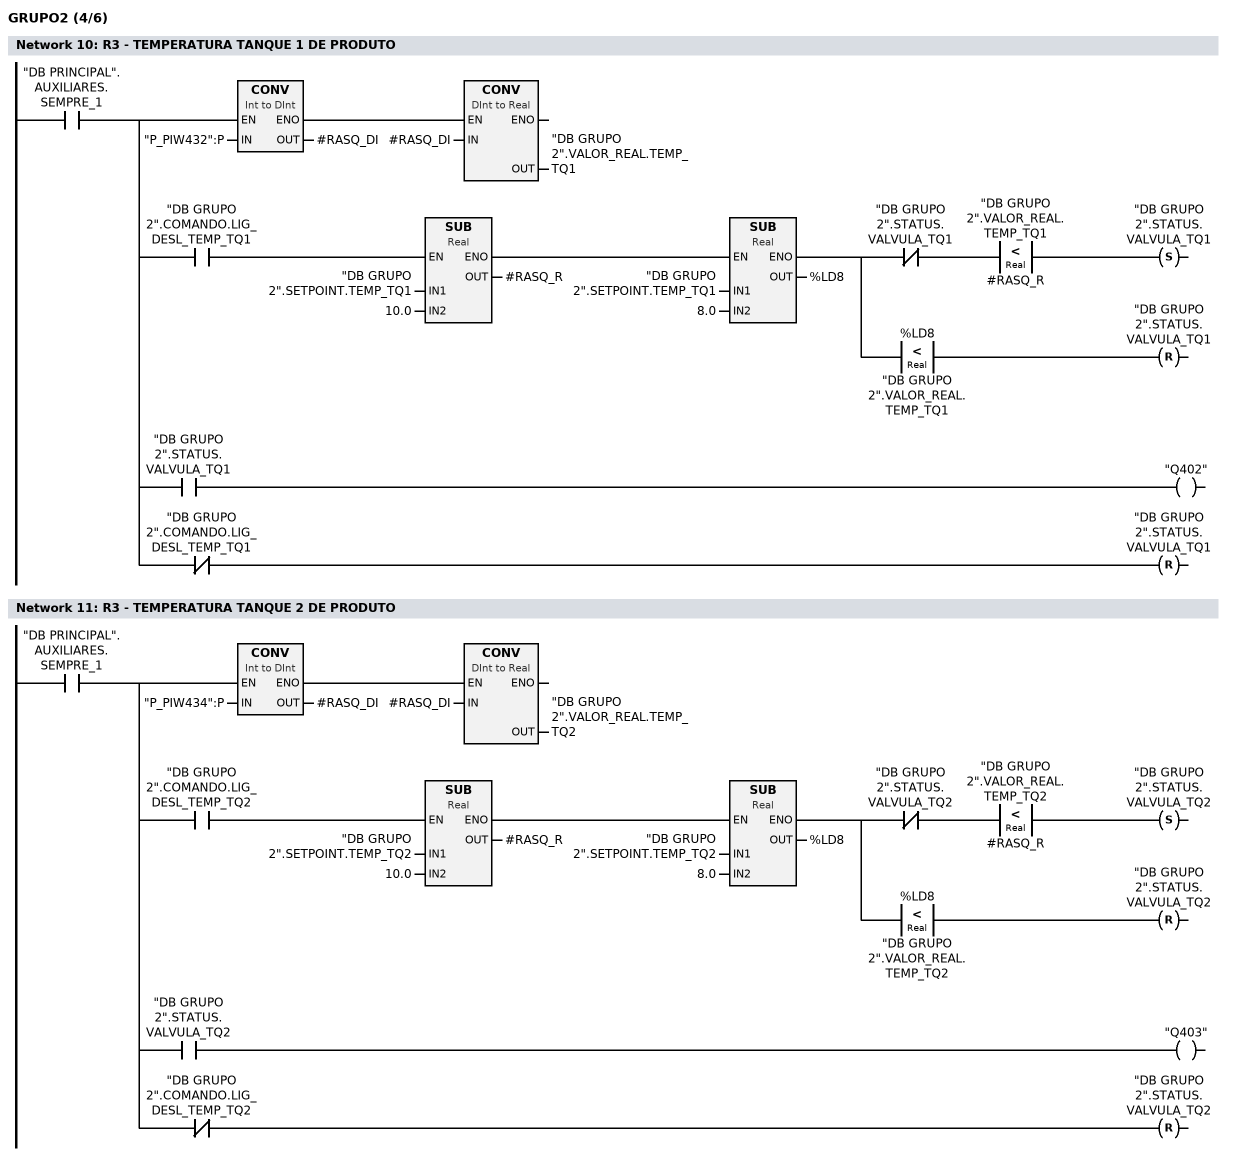
   RUNG wire#powerrail
      Contact( "DB PRINCIPAL".AUXILIARES.SEMPRE_1 )
      wire#w1
      { S7_Templates := "[SrcType := Int, DestType := DInt]"; S7_GenerateENO := "TRUE" } Convert(in := "P_PIW432":P, out => #RASQ_DI)
      { S7_Templates := "[SrcType := DInt, DestType := Real]"; S7_GenerateENO := "TRUE" } Convert(in := #RASQ_DI, out => "DB GRUPO 2".VALOR_REAL.TEMP_TQ1)
   END_RUNG
   RUNG wire#w1
      Contact( "DB GRUPO 2".COMANDO.LIG_DESL_TEMP_TQ1 )
      { S7_Templates := "SrcType := Real"; S7_GenerateENO := "TRUE" } Sub(in1 := "DB GRUPO 2".SETPOINT.TEMP_TQ1, in2 := 10.0, out => #RASQ_R)
      { S7_Templates := "SrcType := Real"; S7_GenerateENO := "TRUE" } Sub(in1 := "DB GRUPO 2".SETPOINT.TEMP_TQ1, in2 := 8.0, out => %LD8)
      wire#w2
      I_Contact( "DB GRUPO 2".STATUS.VALVULA_TQ1 )
      { S7_Templates := "SrcType := Real" } LT_Contact(in1 := "DB GRUPO 2".VALOR_REAL.TEMP_TQ1, in2 := #RASQ_R)
      S_Coil( "DB GRUPO 2".STATUS.VALVULA_TQ1 )
   END_RUNG
   RUNG wire#w2
      { S7_Templates := "SrcType := Real" } LT_Contact(in1 := %LD8, in2 := "DB GRUPO 2".VALOR_REAL.TEMP_TQ1)
      R_Coil( "DB GRUPO 2".STATUS.VALVULA_TQ1 )
   END_RUNG
   RUNG wire#w1
      Contact( "DB GRUPO 2".STATUS.VALVULA_TQ1 )
      Coil( "Q402" )
   END_RUNG
   RUNG wire#w1
      I_Contact( "DB GRUPO 2".COMANDO.LIG_DESL_TEMP_TQ1 )
      R_Coil( "DB GRUPO 2".STATUS.VALVULA_TQ1 )
   END_RUNG
   // the same network as SCL:
   // ENO of a box is taken as its EN; it also drops when the box reports an error
   IF "DB PRINCIPAL".AUXILIARES.SEMPRE_1 THEN
       #RASQ_DI := INT_TO_DINT("P_PIW432":P);
       "DB GRUPO 2".VALOR_REAL.TEMP_TQ1 := DINT_TO_REAL(#RASQ_DI);
   END_IF;
   #_w1 := "DB PRINCIPAL".AUXILIARES.SEMPRE_1 AND "DB GRUPO 2".COMANDO.LIG_DESL_TEMP_TQ1;
   IF #_w1 THEN
       #RASQ_R := "DB GRUPO 2".SETPOINT.TEMP_TQ1 - 10.0;
       %LD8 := "DB GRUPO 2".SETPOINT.TEMP_TQ1 - 8.0;
   END_IF;
   IF #_w1 AND NOT "DB GRUPO 2".STATUS.VALVULA_TQ1 AND ("DB GRUPO 2".VALOR_REAL.TEMP_TQ1 < #RASQ_R) THEN
       "DB GRUPO 2".STATUS.VALVULA_TQ1 := TRUE;
   END_IF;
   IF #_w1 AND (%LD8 < "DB GRUPO 2".VALOR_REAL.TEMP_TQ1) THEN
       "DB GRUPO 2".STATUS.VALVULA_TQ1 := FALSE;
   END_IF;
   "Q402" := "DB PRINCIPAL".AUXILIARES.SEMPRE_1 AND "DB GRUPO 2".STATUS.VALVULA_TQ1;
   IF "DB PRINCIPAL".AUXILIARES.SEMPRE_1 AND NOT "DB GRUPO 2".COMANDO.LIG_DESL_TEMP_TQ1 THEN
       "DB GRUPO 2".STATUS.VALVULA_TQ1 := FALSE;
   END_IF;
END_REGION

REGION Network 11: R3 - TEMPERATURA TANQUE 2 DE PRODUTO
   RUNG wire#powerrail
      Contact( "DB PRINCIPAL".AUXILIARES.SEMPRE_1 )
      wire#w1
      { S7_Templates := "[SrcType := Int, DestType := DInt]"; S7_GenerateENO := "TRUE" } Convert(in := "P_PIW434":P, out => #RASQ_DI)
      { S7_Templates := "[SrcType := DInt, DestType := Real]"; S7_GenerateENO := "TRUE" } Convert(in := #RASQ_DI, out => "DB GRUPO 2".VALOR_REAL.TEMP_TQ2)
   END_RUNG
   RUNG wire#w1
      Contact( "DB GRUPO 2".COMANDO.LIG_DESL_TEMP_TQ2 )
      { S7_Templates := "SrcType := Real"; S7_GenerateENO := "TRUE" } Sub(in1 := "DB GRUPO 2".SETPOINT.TEMP_TQ2, in2 := 10.0, out => #RASQ_R)
      { S7_Templates := "SrcType := Real"; S7_GenerateENO := "TRUE" } Sub(in1 := "DB GRUPO 2".SETPOINT.TEMP_TQ2, in2 := 8.0, out => %LD8)
      wire#w2
      I_Contact( "DB GRUPO 2".STATUS.VALVULA_TQ2 )
      { S7_Templates := "SrcType := Real" } LT_Contact(in1 := "DB GRUPO 2".VALOR_REAL.TEMP_TQ2, in2 := #RASQ_R)
      S_Coil( "DB GRUPO 2".STATUS.VALVULA_TQ2 )
   END_RUNG
   RUNG wire#w2
      { S7_Templates := "SrcType := Real" } LT_Contact(in1 := %LD8, in2 := "DB GRUPO 2".VALOR_REAL.TEMP_TQ2)
      R_Coil( "DB GRUPO 2".STATUS.VALVULA_TQ2 )
   END_RUNG
   RUNG wire#w1
      Contact( "DB GRUPO 2".STATUS.VALVULA_TQ2 )
      Coil( "Q403" )
   END_RUNG
   RUNG wire#w1
      I_Contact( "DB GRUPO 2".COMANDO.LIG_DESL_TEMP_TQ2 )
      R_Coil( "DB GRUPO 2".STATUS.VALVULA_TQ2 )
   END_RUNG
   // the same network as SCL:
   // ENO of a box is taken as its EN; it also drops when the box reports an error
   IF "DB PRINCIPAL".AUXILIARES.SEMPRE_1 THEN
       #RASQ_DI := INT_TO_DINT("P_PIW434":P);
       "DB GRUPO 2".VALOR_REAL.TEMP_TQ2 := DINT_TO_REAL(#RASQ_DI);
   END_IF;
   #_w1 := "DB PRINCIPAL".AUXILIARES.SEMPRE_1 AND "DB GRUPO 2".COMANDO.LIG_DESL_TEMP_TQ2;
   IF #_w1 THEN
       #RASQ_R := "DB GRUPO 2".SETPOINT.TEMP_TQ2 - 10.0;
       %LD8 := "DB GRUPO 2".SETPOINT.TEMP_TQ2 - 8.0;
   END_IF;
   IF #_w1 AND NOT "DB GRUPO 2".STATUS.VALVULA_TQ2 AND ("DB GRUPO 2".VALOR_REAL.TEMP_TQ2 < #RASQ_R) THEN
       "DB GRUPO 2".STATUS.VALVULA_TQ2 := TRUE;
   END_IF;
   IF #_w1 AND (%LD8 < "DB GRUPO 2".VALOR_REAL.TEMP_TQ2) THEN
       "DB GRUPO 2".STATUS.VALVULA_TQ2 := FALSE;
   END_IF;
   "Q403" := "DB PRINCIPAL".AUXILIARES.SEMPRE_1 AND "DB GRUPO 2".STATUS.VALVULA_TQ2;
   IF "DB PRINCIPAL".AUXILIARES.SEMPRE_1 AND NOT "DB GRUPO 2".COMANDO.LIG_DESL_TEMP_TQ2 THEN
       "DB GRUPO 2".STATUS.VALVULA_TQ2 := FALSE;
   END_IF;
END_REGION

REGION Network 12: R3 - TEMPERATURA TANQUE 3 DE PRODUTO
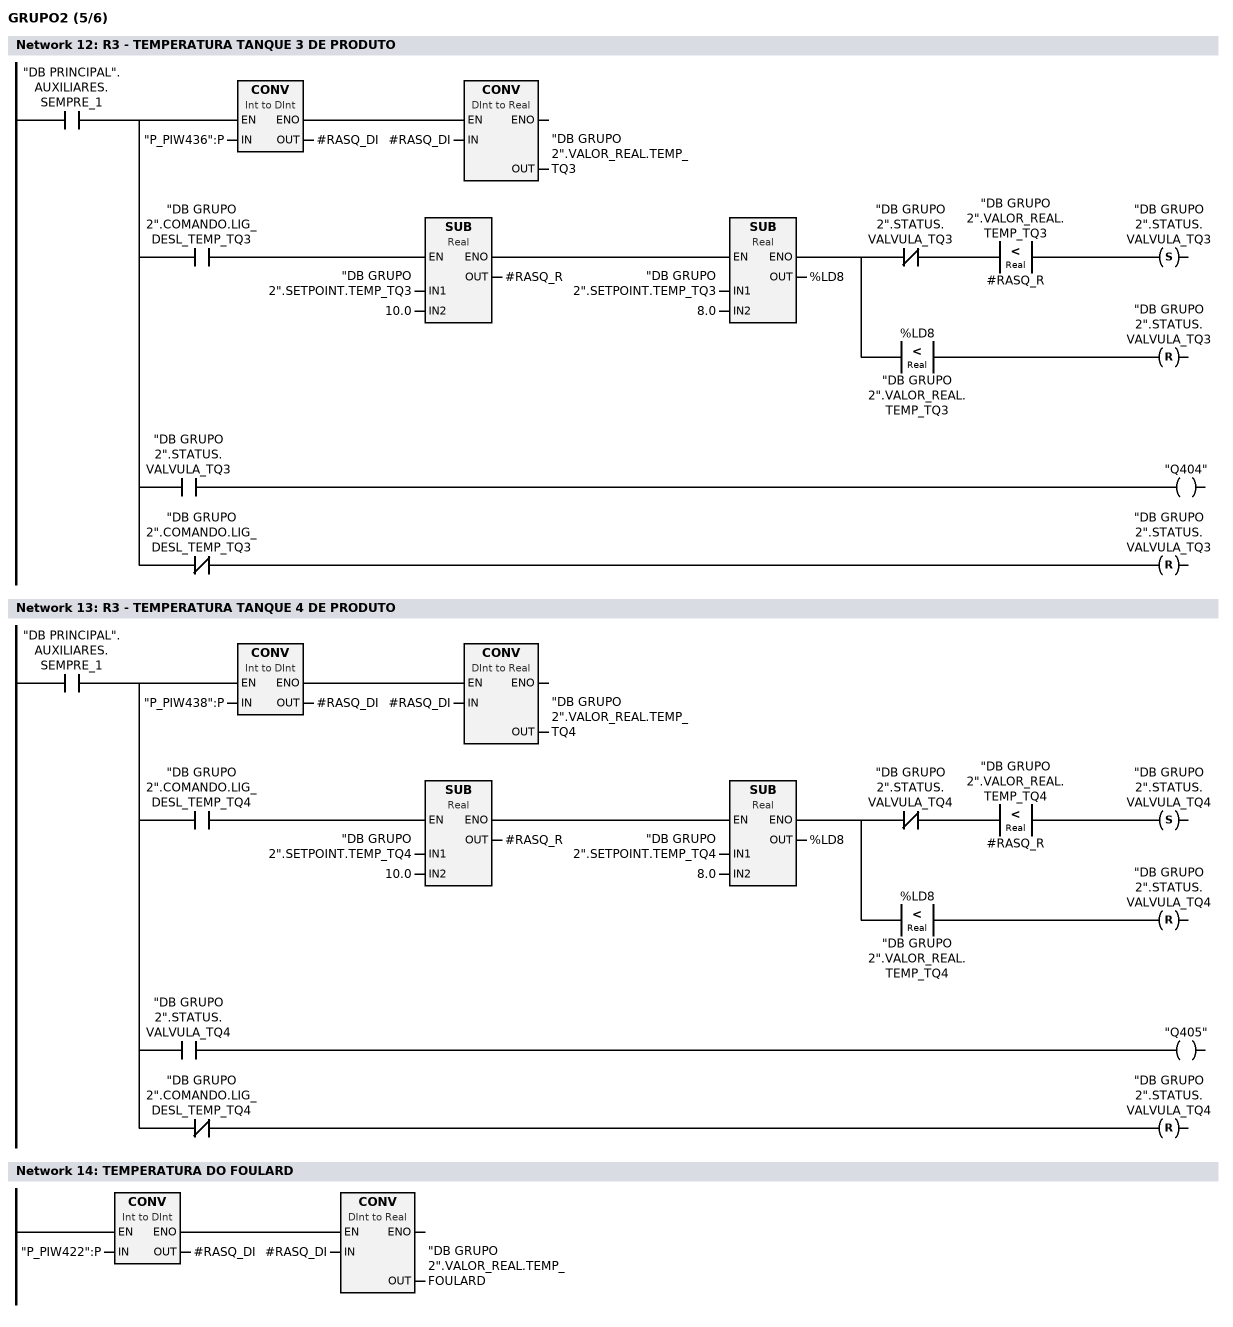
   RUNG wire#powerrail
      Contact( "DB PRINCIPAL".AUXILIARES.SEMPRE_1 )
      wire#w1
      { S7_Templates := "[SrcType := Int, DestType := DInt]"; S7_GenerateENO := "TRUE" } Convert(in := "P_PIW436":P, out => #RASQ_DI)
      { S7_Templates := "[SrcType := DInt, DestType := Real]"; S7_GenerateENO := "TRUE" } Convert(in := #RASQ_DI, out => "DB GRUPO 2".VALOR_REAL.TEMP_TQ3)
   END_RUNG
   RUNG wire#w1
      Contact( "DB GRUPO 2".COMANDO.LIG_DESL_TEMP_TQ3 )
      { S7_Templates := "SrcType := Real"; S7_GenerateENO := "TRUE" } Sub(in1 := "DB GRUPO 2".SETPOINT.TEMP_TQ3, in2 := 10.0, out => #RASQ_R)
      { S7_Templates := "SrcType := Real"; S7_GenerateENO := "TRUE" } Sub(in1 := "DB GRUPO 2".SETPOINT.TEMP_TQ3, in2 := 8.0, out => %LD8)
      wire#w2
      I_Contact( "DB GRUPO 2".STATUS.VALVULA_TQ3 )
      { S7_Templates := "SrcType := Real" } LT_Contact(in1 := "DB GRUPO 2".VALOR_REAL.TEMP_TQ3, in2 := #RASQ_R)
      S_Coil( "DB GRUPO 2".STATUS.VALVULA_TQ3 )
   END_RUNG
   RUNG wire#w2
      { S7_Templates := "SrcType := Real" } LT_Contact(in1 := %LD8, in2 := "DB GRUPO 2".VALOR_REAL.TEMP_TQ3)
      R_Coil( "DB GRUPO 2".STATUS.VALVULA_TQ3 )
   END_RUNG
   RUNG wire#w1
      Contact( "DB GRUPO 2".STATUS.VALVULA_TQ3 )
      Coil( "Q404" )
   END_RUNG
   RUNG wire#w1
      I_Contact( "DB GRUPO 2".COMANDO.LIG_DESL_TEMP_TQ3 )
      R_Coil( "DB GRUPO 2".STATUS.VALVULA_TQ3 )
   END_RUNG
   // the same network as SCL:
   // ENO of a box is taken as its EN; it also drops when the box reports an error
   IF "DB PRINCIPAL".AUXILIARES.SEMPRE_1 THEN
       #RASQ_DI := INT_TO_DINT("P_PIW436":P);
       "DB GRUPO 2".VALOR_REAL.TEMP_TQ3 := DINT_TO_REAL(#RASQ_DI);
   END_IF;
   #_w1 := "DB PRINCIPAL".AUXILIARES.SEMPRE_1 AND "DB GRUPO 2".COMANDO.LIG_DESL_TEMP_TQ3;
   IF #_w1 THEN
       #RASQ_R := "DB GRUPO 2".SETPOINT.TEMP_TQ3 - 10.0;
       %LD8 := "DB GRUPO 2".SETPOINT.TEMP_TQ3 - 8.0;
   END_IF;
   IF #_w1 AND NOT "DB GRUPO 2".STATUS.VALVULA_TQ3 AND ("DB GRUPO 2".VALOR_REAL.TEMP_TQ3 < #RASQ_R) THEN
       "DB GRUPO 2".STATUS.VALVULA_TQ3 := TRUE;
   END_IF;
   IF #_w1 AND (%LD8 < "DB GRUPO 2".VALOR_REAL.TEMP_TQ3) THEN
       "DB GRUPO 2".STATUS.VALVULA_TQ3 := FALSE;
   END_IF;
   "Q404" := "DB PRINCIPAL".AUXILIARES.SEMPRE_1 AND "DB GRUPO 2".STATUS.VALVULA_TQ3;
   IF "DB PRINCIPAL".AUXILIARES.SEMPRE_1 AND NOT "DB GRUPO 2".COMANDO.LIG_DESL_TEMP_TQ3 THEN
       "DB GRUPO 2".STATUS.VALVULA_TQ3 := FALSE;
   END_IF;
END_REGION

REGION Network 13: R3 - TEMPERATURA TANQUE 4 DE PRODUTO
   RUNG wire#powerrail
      Contact( "DB PRINCIPAL".AUXILIARES.SEMPRE_1 )
      wire#w1
      { S7_Templates := "[SrcType := Int, DestType := DInt]"; S7_GenerateENO := "TRUE" } Convert(in := "P_PIW438":P, out => #RASQ_DI)
      { S7_Templates := "[SrcType := DInt, DestType := Real]"; S7_GenerateENO := "TRUE" } Convert(in := #RASQ_DI, out => "DB GRUPO 2".VALOR_REAL.TEMP_TQ4)
   END_RUNG
   RUNG wire#w1
      Contact( "DB GRUPO 2".COMANDO.LIG_DESL_TEMP_TQ4 )
      { S7_Templates := "SrcType := Real"; S7_GenerateENO := "TRUE" } Sub(in1 := "DB GRUPO 2".SETPOINT.TEMP_TQ4, in2 := 10.0, out => #RASQ_R)
      { S7_Templates := "SrcType := Real"; S7_GenerateENO := "TRUE" } Sub(in1 := "DB GRUPO 2".SETPOINT.TEMP_TQ4, in2 := 8.0, out => %LD8)
      wire#w2
      I_Contact( "DB GRUPO 2".STATUS.VALVULA_TQ4 )
      { S7_Templates := "SrcType := Real" } LT_Contact(in1 := "DB GRUPO 2".VALOR_REAL.TEMP_TQ4, in2 := #RASQ_R)
      S_Coil( "DB GRUPO 2".STATUS.VALVULA_TQ4 )
   END_RUNG
   RUNG wire#w2
      { S7_Templates := "SrcType := Real" } LT_Contact(in1 := %LD8, in2 := "DB GRUPO 2".VALOR_REAL.TEMP_TQ4)
      R_Coil( "DB GRUPO 2".STATUS.VALVULA_TQ4 )
   END_RUNG
   RUNG wire#w1
      Contact( "DB GRUPO 2".STATUS.VALVULA_TQ4 )
      Coil( "Q405" )
   END_RUNG
   RUNG wire#w1
      I_Contact( "DB GRUPO 2".COMANDO.LIG_DESL_TEMP_TQ4 )
      R_Coil( "DB GRUPO 2".STATUS.VALVULA_TQ4 )
   END_RUNG
   // the same network as SCL:
   // ENO of a box is taken as its EN; it also drops when the box reports an error
   IF "DB PRINCIPAL".AUXILIARES.SEMPRE_1 THEN
       #RASQ_DI := INT_TO_DINT("P_PIW438":P);
       "DB GRUPO 2".VALOR_REAL.TEMP_TQ4 := DINT_TO_REAL(#RASQ_DI);
   END_IF;
   #_w1 := "DB PRINCIPAL".AUXILIARES.SEMPRE_1 AND "DB GRUPO 2".COMANDO.LIG_DESL_TEMP_TQ4;
   IF #_w1 THEN
       #RASQ_R := "DB GRUPO 2".SETPOINT.TEMP_TQ4 - 10.0;
       %LD8 := "DB GRUPO 2".SETPOINT.TEMP_TQ4 - 8.0;
   END_IF;
   IF #_w1 AND NOT "DB GRUPO 2".STATUS.VALVULA_TQ4 AND ("DB GRUPO 2".VALOR_REAL.TEMP_TQ4 < #RASQ_R) THEN
       "DB GRUPO 2".STATUS.VALVULA_TQ4 := TRUE;
   END_IF;
   IF #_w1 AND (%LD8 < "DB GRUPO 2".VALOR_REAL.TEMP_TQ4) THEN
       "DB GRUPO 2".STATUS.VALVULA_TQ4 := FALSE;
   END_IF;
   "Q405" := "DB PRINCIPAL".AUXILIARES.SEMPRE_1 AND "DB GRUPO 2".STATUS.VALVULA_TQ4;
   IF "DB PRINCIPAL".AUXILIARES.SEMPRE_1 AND NOT "DB GRUPO 2".COMANDO.LIG_DESL_TEMP_TQ4 THEN
       "DB GRUPO 2".STATUS.VALVULA_TQ4 := FALSE;
   END_IF;
END_REGION

REGION Network 14: TEMPERATURA DO FOULARD
   RUNG wire#powerrail
      { S7_Templates := "[SrcType := Int, DestType := DInt]"; S7_GenerateENO := "TRUE" } Convert(in := "P_PIW422":P, out => #RASQ_DI)
      { S7_Templates := "[SrcType := DInt, DestType := Real]"; S7_GenerateENO := "TRUE" } Convert(in := #RASQ_DI, out => "DB GRUPO 2".VALOR_REAL.TEMP_FOULARD)
   END_RUNG
   // the same network as SCL:
   // ENO of a box is taken as its EN; it also drops when the box reports an error
   #RASQ_DI := INT_TO_DINT("P_PIW422":P);
   "DB GRUPO 2".VALOR_REAL.TEMP_FOULARD := DINT_TO_REAL(#RASQ_DI);
END_REGION

REGION Network 15
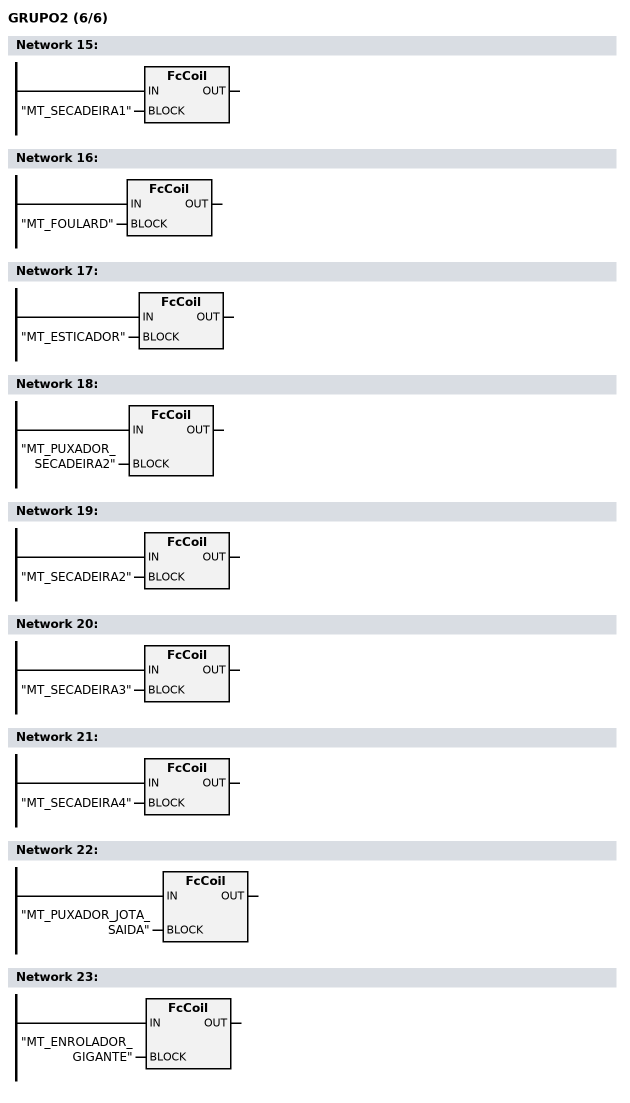
   // no SCL statement known for FcCoil: written as a call
   FcCoil(block := "MT_SECADEIRA1", in := TRUE);
END_REGION

REGION Network 16
   // no SCL statement known for FcCoil: written as a call
   FcCoil(block := "MT_FOULARD", in := TRUE);
END_REGION

REGION Network 17
   // no SCL statement known for FcCoil: written as a call
   FcCoil(block := "MT_ESTICADOR", in := TRUE);
END_REGION

REGION Network 18
   // no SCL statement known for FcCoil: written as a call
   FcCoil(block := "MT_PUXADOR_SECADEIRA2", in := TRUE);
END_REGION

REGION Network 19
   // no SCL statement known for FcCoil: written as a call
   FcCoil(block := "MT_SECADEIRA2", in := TRUE);
END_REGION

REGION Network 20
   // no SCL statement known for FcCoil: written as a call
   FcCoil(block := "MT_SECADEIRA3", in := TRUE);
END_REGION

REGION Network 21
   // no SCL statement known for FcCoil: written as a call
   FcCoil(block := "MT_SECADEIRA4", in := TRUE);
END_REGION

REGION Network 22
   // no SCL statement known for FcCoil: written as a call
   FcCoil(block := "MT_PUXADOR_JOTA_SAIDA", in := TRUE);
END_REGION

REGION Network 23
   // no SCL statement known for FcCoil: written as a call
   FcCoil(block := "MT_ENROLADOR_GIGANTE", in := TRUE);
END_REGION
END_FUNCTION

FUNCTION "PID" : Void   // FC7, LAD
TITLE = MÓDULO DE CONTROLE DE TEMPERATURAS
{ S7_Optimized_Access := 'FALSE' }
VERSION : 0.1
// DATA BLOCK DE CONTROLE // DB7
// Automation Pack Automação Indl. e Com. Ltda.
// Cliente: Texima S/A Ind. de Máquinas
// Cliente Final: CEDRO TEXTIL
// Máquina: Linha 1 - O.S.: 24.626
   VAR_TEMP
      RASCUNHO_INT_1 : Int;   // RASCUNHO
      RASCUNHO_WORD_2 : Word;   // RASCUNHO
      RASCUNHO_DINT_1 : DInt;   // RASCUNHO
      RASCUNHO_DINT_2 : DInt;   // RASCUNHO
      RASCUNHO_REAL_1 : Real;   // RASCUNHO
      RASCUNHO_REAL_2 : Real;   // RASCUNHO
   END_VAR
   VAR_TEMP   // added for the SCL form of the ladder/FBD networks
      _w1 : Bool;
   END_VAR
BEGIN

REGION Network 1
   // NEUTRALIZACAO 1
